LIN {X 0,Y 143.297,Z 453.566,A -85,B 0,C 180,E1 -24317.114,E2 -24317.114} C_VEL
LIN {X 0,Y 143.279,Z 453.631,A -85,B 0,C 180,E1 -24321.255,E2 -24321.255} C_VEL
LIN {X 0,Y 143.191,Z 453.587,A -85,B 0,C 180,E1 -24327.936,E2 -24327.936} C_VEL
LIN {X 0,Y 143.153,Z 453.64,A -85,B 0,C 180,E1 -24331.545,E2 -24331.545} C_VEL
LIN {X 0,Y 144.077,Z 456.331,A -85,B 0,C 180,E1 -24332.694,E2 -24332.694} C_VEL
LIN {X 0,Y 146.083,Z 458.522,A -85,B 0,C 180,E1 -24334.465,E2 -24334.465} C_VEL
LIN {X 0,Y 146.787,Z 459.324,A -85,B 0,C 180,E1 -24335.068,E2 -24335.068} C_VEL
LIN {X 0,Y 148.061,Z 461.946,A -85,B 0,C 180,E1 -24336.393,E2 -24336.393} C_VEL
LIN {X 0,Y 149.588,Z 463.631,A -85,B 0,C 180,E1 -24337.646,E2 -24337.646} C_VEL
LIN {X 0,Y 151.047,Z 466.609,A -85,B 0,C 180,E1 -24339.128,E2 -24339.128} C_VEL
LIN {X 0,Y 154.334,Z 472.293,A -85,B 0,C 180,E1 -24342.197,E2 -24342.197} C_VEL
LIN {X 0,Y 157.932,Z 480.262,A -85,B 0,C 180,E1 -24346.023,E2 -24346.023} C_VEL
LIN {X 0,Y 160.847,Z 488.732,A -85,B 0,C 180,E1 -24349.874,E2 -24349.874} C_VEL
LIN {X 0,Y 162.593,Z 495.92,A -85,B 0,C 180,E1 -24353.096,E2 -24353.096} C_VEL
LIN {X 0,Y 163.683,Z 502.348,A -85,B 0,C 180,E1 -24356.07,E2 -24356.07} C_VEL
LIN {X 0,Y 163.818,Z 503.973,A -85,B 0,C 180,E1 -24356.839,E2 -24356.839} C_VEL
LIN {X 0,Y 161.807,Z 508.944,A -85,B 0,C 180,E1 -24358.586,E2 -24358.586} C_VEL
LIN {X 0,Y 157.646,Z 517.43,A -85,B 0,C 180,E1 -24362.089,E2 -24362.089} C_VEL
LIN {X 0,Y 153.752,Z 524.699,A -85,B 0,C 180,E1 -24366.093,E2 -24366.093} C_VEL
LIN {X 0,Y 151.144,Z 529.533,A -85,B 0,C 180,E1 -24369.589,E2 -24369.589} C_VEL
LIN {X 0,Y 148.515,Z 533.769,A -85,B 0,C 180,E1 -24373.505,E2 -24373.505} C_VEL
LIN {X 0,Y 147.12,Z 536.002,A -85,B 0,C 180,E1 -24376.181,E2 -24376.181} C_VEL
LIN {X 0,Y 145.943,Z 537.821,A -85,B 0,C 180,E1 -24378.894,E2 -24378.894} C_VEL
LIN {X 0,Y 145.02,Z 539.188,A -85,B 0,C 180,E1 -24381.64,E2 -24381.64} C_VEL
LIN {X 0,Y 144.307,Z 540.706,A -85,B 0,C 180,E1 -24387.208,E2 -24387.208} C_VEL
LIN {X 0,Y 144.213,Z 540.925,A -85,B 0,C 180,E1 -24390,E2 -24390} C_VEL
LIN {X 0,Y 144.306,Z 540.736,A -85,B 0,C 180,E1 -24392.791,E2 -24392.791} C_VEL
LIN {X 0,Y 145.009,Z 539.256,A -85,B 0,C 180,E1 -24398.36,E2 -24398.36} C_VEL
LIN {X 0,Y 145.924,Z 537.921,A -85,B 0,C 180,E1 -24401.107,E2 -24401.107} C_VEL
LIN {X 0,Y 147.831,Z 535.093,A -85,B 0,C 180,E1 -24405.157,E2 -24405.157} C_VEL
LIN {X 0,Y 150.232,Z 531.269,A -85,B 0,C 180,E1 -24409.115,E2 -24409.115} C_VEL
LIN {X 0,Y 153.482,Z 525.332,A -85,B 0,C 180,E1 -24413.679,E2 -24413.679} C_VEL
LIN {X 0,Y 157.622,Z 517.742,A -85,B 0,C 180,E1 -24417.915,E2 -24417.915} C_VEL
LIN {X 0,Y 161.738,Z 509.36,A -85,B 0,C 180,E1 -24421.429,E2 -24421.429} C_VEL
LIN {X 0,Y 163.827,Z 504.413,A -85,B 0,C 180,E1 -24423.159,E2 -24423.159} C_VEL
LIN {X 0,Y 163.074,Z 497.829,A -85,B 0,C 180,E1 -24426.2,E2 -24426.2} C_VEL
LIN {X 0,Y 161.008,Z 488.99,A -85,B 0,C 180,E1 -24430.194,E2 -24430.194} C_VEL
LIN {X 0,Y 158.209,Z 480.766,A -85,B 0,C 180,E1 -24433.939,E2 -24433.939} C_VEL
LIN {X 0,Y 154.527,Z 472.644,A -85,B 0,C 180,E1 -24437.868,E2 -24437.868} C_VEL
LIN {X 0,Y 149.779,Z 464.121,A -85,B 0,C 180,E1 -24442.411,E2 -24442.411} C_VEL
LIN {X 0,Y 147.619,Z 461.218,A -85,B 0,C 180,E1 -24444.324,E2 -24444.324} C_VEL
LIN {X 0,Y 146.552,Z 458.872,A -85,B 0,C 180,E1 -24445.463,E2 -24445.463} C_VEL
LIN {X 0,Y 144.33,Z 456.714,A -85,B 0,C 180,E1 -24447.371,E2 -24447.371} C_VEL
LIN {X 0,Y 143.255,Z 454.252,A -85,B 0,C 180,E1 -24448.583,E2 -24448.583} C_VEL
LIN {X 0,Y 143.158,Z 453.648,A -85,B 0,C 180,E1 -24448.868,E2 -24448.868} C_VEL
LIN {X 0,Y 143.161,Z 453.647,A -85,B 0,C 180,E1 -24453.779,E2 -24453.779} C_VEL
LIN {X 0,Y 143.311,Z 453.634,A -85,B 0,C 180,E1 -24459.923,E2 -24459.923} C_VEL
LIN {X 0,Y 143.364,Z 453.627,A -85,B 0,C 180,E1 -24465.811,E2 -24465.811} C_VEL
LIN {X 0,Y 143.539,Z 453.594,A -85,B 0,C 180,E1 -24468.705,E2 -24468.705} C_VEL
LIN {X 0,Y 143.627,Z 453.594,A -85,B 0,C 180,E1 -24471.558,E2 -24471.558} C_VEL
LIN {X 0,Y 144.179,Z 453.515,A -85,B 0,C 180,E1 -24480,E2 -24480} C_VEL
LIN {X 0,Y 143.627,Z 453.581,A -85,B 0,C 180,E1 -24488.441,E2 -24488.441} C_VEL
LIN {X 0,Y 143.507,Z 453.601,A -85,B 0,C 180,E1 -24491.631,E2 -24491.631} C_VEL
LIN {X 0,Y 143.349,Z 453.727,A -85,B 0,C 180,E1 -24494.552,E2 -24494.552} C_VEL
LIN {X 0,Y 143.984,Z 456.816,A -85,B 0,C 180,E1 -24499.979,E2 -24499.979} C_VEL
LIN {X 0,Y 145.063,Z 461.745,A -85,B 0,C 180,E1 -24507.404,E2 -24507.404} C_VEL
LIN {X 0,Y 145.674,Z 465.026,A -85,B 0,C 180,E1 -24511.456,E2 -24511.456} C_VEL
LIN {X 0,Y 147.336,Z 468.84,A -85,B 0,C 180,E1 -24512.86,E2 -24512.86} C_VEL
LIN {X 0,Y 149.667,Z 472.325,A -85,B 0,C 180,E1 -24514.58,E2 -24514.58} C_VEL
LIN {X 0,Y 151.366,Z 476.461,A -85,B 0,C 180,E1 -24515.989,E2 -24515.989} C_VEL
LIN {X 0,Y 152.885,Z 479.225,A -85,B 0,C 180,E1 -24517.11,E2 -24517.11} C_VEL
LIN {X 0,Y 155.096,Z 484.217,A -85,B 0,C 180,E1 -24518.852,E2 -24518.852} C_VEL
LIN {X 0,Y 159.394,Z 496.028,A -85,B 0,C 180,E1 -24522.582,E2 -24522.582} C_VEL
LIN {X 0,Y 159.768,Z 503.297,A -85,B 0,C 180,E1 -24524.191,E2 -24524.191} C_VEL
LIN {X 0,Y 159.384,Z 515.58,A -85,B 0,C 180,E1 -24527.018,E2 -24527.018} C_VEL
LIN {X 0,Y 158.225,Z 526.386,A -85,B 0,C 180,E1 -24529.818,E2 -24529.818} C_VEL
LIN {X 0,Y 156.296,Z 537.075,A -85,B 0,C 180,E1 -24533.028,E2 -24533.028} C_VEL
LIN {X 0,Y 154.059,Z 545.932,A -85,B 0,C 180,E1 -24536.151,E2 -24536.151} C_VEL
LIN {X 0,Y 151.298,Z 555.019,A -85,B 0,C 180,E1 -24540.043,E2 -24540.043} C_VEL
LIN {X 0,Y 148.719,Z 561.324,A -85,B 0,C 180,E1 -24543.324,E2 -24543.324} C_VEL
LIN {X 0,Y 145.685,Z 567.48,A -85,B 0,C 180,E1 -24547.299,E2 -24547.299} C_VEL
LIN {X 0,Y 143.571,Z 572.416,A -85,B 0,C 180,E1 -24551.447,E2 -24551.447} C_VEL
LIN {X 0,Y 142.375,Z 576.263,A -85,B 0,C 180,E1 -24555.711,E2 -24555.711} C_VEL
LIN {X 0,Y 142.003,Z 578.283,A -85,B 0,C 180,E1 -24558.582,E2 -24558.582} C_VEL
LIN {X 0,Y 142.305,Z 580.995,A -85,B 0,C 180,E1 -24564.332,E2 -24564.332} C_VEL
LIN {X 0,Y 142.75,Z 581.734,A -85,B 0,C 180,E1 -24567.178,E2 -24567.178} C_VEL
LIN {X 0,Y 143.416,Z 582.062,A -85,B 0,C 180,E1 -24570,E2 -24570} C_VEL
LIN {X 0,Y 142.744,Z 581.719,A -85,B 0,C 180,E1 -24572.822,E2 -24572.822} C_VEL
LIN {X 0,Y 142.297,Z 580.972,A -85,B 0,C 180,E1 -24575.669,E2 -24575.669} C_VEL
LIN {X 0,Y 142.004,Z 579.81,A -85,B 0,C 180,E1 -24578.539,E2 -24578.539} C_VEL
LIN {X 0,Y 142.155,Z 577.262,A -85,B 0,C 180,E1 -24582.855,E2 -24582.855} C_VEL
LIN {X 0,Y 143.044,Z 573.723,A -85,B 0,C 180,E1 -24587.145,E2 -24587.145} C_VEL
LIN {X 0,Y 144.83,Z 569.135,A -85,B 0,C 180,E1 -24591.343,E2 -24591.343} C_VEL
LIN {X 0,Y 148.156,Z 562.333,A -85,B 0,C 180,E1 -24596.027,E2 -24596.027} C_VEL
LIN {X 0,Y 150.773,Z 556.234,A -85,B 0,C 180,E1 -24599.304,E2 -24599.304} C_VEL
LIN {X 0,Y 153.633,Z 547.156,A -85,B 0,C 180,E1 -24603.295,E2 -24603.295} C_VEL
LIN {X 0,Y 156,Z 537.835,A -85,B 0,C 180,E1 -24606.651,E2 -24606.651} C_VEL
LIN {X 0,Y 157.978,Z 527.397,A -85,B 0,C 180,E1 -24609.814,E2 -24609.814} C_VEL
LIN {X 0,Y 159.187,Z 516.722,A -85,B 0,C 180,E1 -24612.626,E2 -24612.626} C_VEL
LIN {X 0,Y 159.693,Z 504.397,A -85,B 0,C 180,E1 -24615.481,E2 -24615.481} C_VEL
LIN {X 0,Y 159.493,Z 497.348,A -85,B 0,C 180,E1 -24617.002,E2 -24617.002} C_VEL
LIN {X 0,Y 158.812,Z 494.119,A -85,B 0,C 180,E1 -24617.868,E2 -24617.868} C_VEL
LIN {X 0,Y 154.735,Z 483.639,A -85,B 0,C 180,E1 -24621.249,E2 -24621.249} C_VEL
LIN {X 0,Y 153.2,Z 480.223,A -85,B 0,C 180,E1 -24622.45,E2 -24622.45} C_VEL
LIN {X 0,Y 152.039,Z 477.482,A -85,B 0,C 180,E1 -24623.379,E2 -24623.379} C_VEL
LIN {X 0,Y 150.429,Z 475.392,A -85,B 0,C 180,E1 -24624.466,E2 -24624.466} C_VEL
LIN {X 0,Y 146.597,Z 472.525,A -85,B 0,C 180,E1 -24626.916,E2 -24626.916} C_VEL
LIN {X 0,Y 142.658,Z 470.103,A -85,B 0,C 180,E1 -24629.618,E2 -24629.618} C_VEL
LIN {X 0,Y 140.203,Z 467.568,A -85,B 0,C 180,E1 -24631.637,E2 -24631.637} C_VEL
LIN {X 0,Y 139.55,Z 466.445,A -85,B 0,C 180,E1 -24632.278,E2 -24632.278} C_VEL
LIN {X 0,Y 137.989,Z 462.532,A -85,B 0,C 180,E1 -24634.145,E2 -24634.145} C_VEL
LIN {X 0,Y 137.296,Z 459.461,A -85,B 0,C 180,E1 -24639.003,E2 -24639.003} C_VEL
LIN {X 0,Y 136.944,Z 457.668,A -85,B 0,C 180,E1 -24642.066,E2 -24642.066} C_VEL
LIN {X 0,Y 136.47,Z 454.488,A -85,B 0,C 180,E1 -24648.387,E2 -24648.387} C_VEL
LIN {X 0,Y 136.554,Z 454.477,A -85,B 0,C 180,E1 -24651.118,E2 -24651.118} C_VEL
LIN {X 0,Y 137.137,Z 454.4,A -85,B 0,C 180,E1 -24660,E2 -24660} C_VEL
LIN {X 0,Y 136.554,Z 454.476,A -85,B 0,C 180,E1 -24668.882,E2 -24668.882} C_VEL
LIN {X 0,Y 136.443,Z 454.448,A -85,B 0,C 180,E1 -24671.89,E2 -24671.89} C_VEL
LIN {X 0,Y 136.215,Z 454.454,A -85,B 0,C 180,E1 -24678.034,E2 -24678.034} C_VEL
LIN {X 0,Y 136.2,Z 454.515,A -85,B 0,C 180,E1 -24681.749,E2 -24681.749} C_VEL
LIN {X 0,Y 136.123,Z 454.518,A -85,B 0,C 180,E1 -24686.031,E2 -24686.031} C_VEL
LIN {X 0,Y 136.969,Z 457.004,A -85,B 0,C 180,E1 -24687.4,E2 -24687.4} C_VEL
LIN {X 0,Y 138.795,Z 459.225,A -85,B 0,C 180,E1 -24689.47,E2 -24689.47} C_VEL
LIN {X 0,Y 139.999,Z 460.171,A -85,B 0,C 180,E1 -24690.654,E2 -24690.654} C_VEL
LIN {X 0,Y 141.216,Z 462.885,A -85,B 0,C 180,E1 -24692.214,E2 -24692.214} C_VEL
LIN {X 0,Y 143.317,Z 465.418,A -85,B 0,C 180,E1 -24694.329,E2 -24694.329} C_VEL
LIN {X 0,Y 144.49,Z 467.805,A -85,B 0,C 180,E1 -24695.71,E2 -24695.71} C_VEL
LIN {X 0,Y 145.415,Z 468.906,A -85,B 0,C 180,E1 -24696.586,E2 -24696.586} C_VEL
LIN {X 0,Y 150.05,Z 477.982,A -85,B 0,C 180,E1 -24701.779,E2 -24701.779} C_VEL
LIN {X 0,Y 152.992,Z 485.164,A -85,B 0,C 180,E1 -24705.508,E2 -24705.508} C_VEL
LIN {X 0,Y 155.326,Z 492.952,A -85,B 0,C 180,E1 -24709.323,E2 -24709.323} C_VEL
LIN {X 0,Y 156.807,Z 500.167,A -85,B 0,C 180,E1 -24712.836,E2 -24712.836} C_VEL
LIN {X 0,Y 157.46,Z 505.072,A -85,B 0,C 180,E1 -24715.314,E2 -24715.314} C_VEL
LIN {X 0,Y 157.385,Z 506.694,A -85,B 0,C 180,E1 -24716.069,E2 -24716.069} C_VEL
LIN {X 0,Y 153.607,Z 514.435,A -85,B 0,C 180,E1 -24719.021,E2 -24719.021} C_VEL
LIN {X 0,Y 149.493,Z 521.994,A -85,B 0,C 180,E1 -24722.718,E2 -24722.718} C_VEL
LIN {X 0,Y 146.667,Z 527.077,A -85,B 0,C 180,E1 -24725.932,E2 -24725.932} C_VEL
LIN {X 0,Y 143.655,Z 532.088,A -85,B 0,C 180,E1 -24729.973,E2 -24729.973} C_VEL
LIN {X 0,Y 141.075,Z 535.962,A -85,B 0,C 180,E1 -24734.097,E2 -24734.097} C_VEL
LIN {X 0,Y 139.053,Z 538.827,A -85,B 0,C 180,E1 -24738.336,E2 -24738.336} C_VEL
LIN {X 0,Y 138.07,Z 540.193,A -85,B 0,C 180,E1 -24741.216,E2 -24741.216} C_VEL
LIN {X 0,Y 137.288,Z 541.712,A -85,B 0,C 180,E1 -24747.065,E2 -24747.065} C_VEL
LIN {X 0,Y 137.186,Z 541.93,A -85,B 0,C 180,E1 -24750,E2 -24750} C_VEL
LIN {X 0,Y 137.287,Z 541.741,A -85,B 0,C 180,E1 -24752.934,E2 -24752.934} C_VEL
LIN {X 0,Y 138.059,Z 540.261,A -85,B 0,C 180,E1 -24758.784,E2 -24758.784} C_VEL
LIN {X 0,Y 139.034,Z 538.925,A -85,B 0,C 180,E1 -24761.665,E2 -24761.665} C_VEL
LIN {X 0,Y 141.06,Z 536.097,A -85,B 0,C 180,E1 -24765.904,E2 -24765.904} C_VEL
LIN {X 0,Y 143.61,Z 532.273,A -85,B 0,C 180,E1 -24770.033,E2 -24770.033} C_VEL
LIN {X 0,Y 147.073,Z 526.335,A -85,B 0,C 180,E1 -24774.779,E2 -24774.779} C_VEL
LIN {X 0,Y 151.448,Z 518.745,A -85,B 0,C 180,E1 -24779.16,E2 -24779.16} C_VEL
LIN {X 0,Y 155.787,Z 510.362,A -85,B 0,C 180,E1 -24782.776,E2 -24782.776} C_VEL
LIN {X 0,Y 157.316,Z 507.142,A -85,B 0,C 180,E1 -24783.947,E2 -24783.947} C_VEL
LIN {X 0,Y 157.546,Z 505.493,A -85,B 0,C 180,E1 -24784.664,E2 -24784.664} C_VEL
LIN {X 0,Y 156.753,Z 499.46,A -85,B 0,C 180,E1 -24787.7,E2 -24787.7} C_VEL
LIN {X 0,Y 155.031,Z 491.486,A -85,B 0,C 180,E1 -24791.583,E2 -24791.583} C_VEL
LIN {X 0,Y 153.006,Z 485.082,A -85,B 0,C 180,E1 -24794.754,E2 -24794.754} C_VEL
LIN {X 0,Y 149.992,Z 477.795,A -85,B 0,C 180,E1 -24798.564,E2 -24798.564} C_VEL
LIN {X 0,Y 146.032,Z 470.057,A -85,B 0,C 180,E1 -24803.018,E2 -24803.018} C_VEL
LIN {X 0,Y 143.522,Z 465.868,A -85,B 0,C 180,E1 -24805.727,E2 -24805.727} C_VEL
LIN {X 0,Y 140.452,Z 461.398,A -85,B 0,C 180,E1 -24809.037,E2 -24809.037} C_VEL
LIN {X 0,Y 139.876,Z 459.943,A -85,B 0,C 180,E1 -24809.838,E2 -24809.838} C_VEL
LIN {X 0,Y 137.633,Z 458.023,A -85,B 0,C 180,E1 -24812.159,E2 -24812.159} C_VEL
LIN {X 0,Y 136.391,Z 455.702,A -85,B 0,C 180,E1 -24813.818,E2 -24813.818} C_VEL
LIN {X 0,Y 136.11,Z 454.53,A -85,B 0,C 180,E1 -24814.48,E2 -24814.48} C_VEL
LIN {X 0,Y 136.246,Z 454.506,A -85,B 0,C 180,E1 -24818.833,E2 -24818.833} C_VEL
LIN {X 0,Y 136.274,Z 454.509,A -85,B 0,C 180,E1 -24825.056,E2 -24825.056} C_VEL
LIN {X 0,Y 136.446,Z 454.477,A -85,B 0,C 180,E1 -24828.138,E2 -24828.138} C_VEL
LIN {X 0,Y 136.553,Z 454.476,A -85,B 0,C 180,E1 -24831.118,E2 -24831.118} C_VEL
LIN {X 0,Y 137.136,Z 454.392,A -85,B 0,C 180,E1 -24840,E2 -24840} C_VEL
LIN {X 0,Y 136.553,Z 454.463,A -85,B 0,C 180,E1 -24848.882,E2 -24848.882} C_VEL
LIN {X 0,Y 136.459,Z 454.644,A -85,B 0,C 180,E1 -24851.889,E2 -24851.889} C_VEL
LIN {X 0,Y 136.954,Z 457.794,A -85,B 0,C 180,E1 -24857.933,E2 -24857.933} C_VEL
LIN {X 0,Y 137.658,Z 461.515,A -85,B 0,C 180,E1 -24864.106,E2 -24864.106} C_VEL
LIN {X 0,Y 137.986,Z 462.686,A -85,B 0,C 180,E1 -24865.755,E2 -24865.755} C_VEL
LIN {X 0,Y 139.872,Z 466.922,A -85,B 0,C 180,E1 -24867.797,E2 -24867.797} C_VEL
LIN {X 0,Y 142.506,Z 470.812,A -85,B 0,C 180,E1 -24870.205,E2 -24870.205} C_VEL
LIN {X 0,Y 144.675,Z 475.595,A -85,B 0,C 180,E1 -24872.3,E2 -24872.3} C_VEL
LIN {X 0,Y 145.984,Z 477.81,A -85,B 0,C 180,E1 -24873.41,E2 -24873.41} C_VEL
LIN {X 0,Y 148.138,Z 482.859,A -85,B 0,C 180,E1 -24875.429,E2 -24875.429} C_VEL
LIN {X 0,Y 152.267,Z 493.635,A -85,B 0,C 180,E1 -24879.393,E2 -24879.393} C_VEL
LIN {X 0,Y 154.104,Z 499.441,A -85,B 0,C 180,E1 -24881.362,E2 -24881.362} C_VEL
LIN {X 0,Y 154.051,Z 508.443,A -85,B 0,C 180,E1 -24883.509,E2 -24883.509} C_VEL
LIN {X 0,Y 153.152,Z 520.101,A -85,B 0,C 180,E1 -24886.502,E2 -24886.502} C_VEL
LIN {X 0,Y 151.471,Z 530.47,A -85,B 0,C 180,E1 -24889.49,E2 -24889.49} C_VEL
LIN {X 0,Y 149.045,Z 540.984,A -85,B 0,C 180,E1 -24893.054,E2 -24893.054} C_VEL
LIN {X 0,Y 146.412,Z 549.526,A -85,B 0,C 180,E1 -24896.494,E2 -24896.494} C_VEL
LIN {X 0,Y 143.945,Z 556.643,A -85,B 0,C 180,E1 -24899.97,E2 -24899.97} C_VEL
LIN {X 0,Y 141.209,Z 562.506,A -85,B 0,C 180,E1 -24903.389,E2 -24903.389} C_VEL
LIN {X 0,Y 138.208,Z 568.218,A -85,B 0,C 180,E1 -24907.581,E2 -24907.581} C_VEL
LIN {X 0,Y 136.211,Z 572.776,A -85,B 0,C 180,E1 -24911.966,E2 -24911.966} C_VEL
LIN {X 0,Y 135.168,Z 576.288,A -85,B 0,C 180,E1 -24916.469,E2 -24916.469} C_VEL
LIN {X 0,Y 134.957,Z 579.099,A -85,B 0,C 180,E1 -24921.667,E2 -24921.667} C_VEL
LIN {X 0,Y 135.667,Z 580.72,A -85,B 0,C 180,E1 -24927.031,E2 -24927.031} C_VEL
LIN {X 0,Y 136.333,Z 581.049,A -85,B 0,C 180,E1 -24930,E2 -24930} C_VEL
LIN {X 0,Y 135.66,Z 580.704,A -85,B 0,C 180,E1 -24932.97,E2 -24932.97} C_VEL
LIN {X 0,Y 134.96,Z 579.063,A -85,B 0,C 180,E1 -24938.342,E2 -24938.342} C_VEL
LIN {X 0,Y 135.168,Z 576.235,A -85,B 0,C 180,E1 -24943.532,E2 -24943.532} C_VEL
LIN {X 0,Y 136.2,Z 572.695,A -85,B 0,C 180,E1 -24948.036,E2 -24948.036} C_VEL
LIN {X 0,Y 138.184,Z 568.109,A -85,B 0,C 180,E1 -24952.424,E2 -24952.424} C_VEL
LIN {X 0,Y 141.208,Z 562.376,A -85,B 0,C 180,E1 -24956.612,E2 -24956.612} C_VEL
LIN {X 0,Y 143.929,Z 556.48,A -85,B 0,C 180,E1 -24960.034,E2 -24960.034} C_VEL
LIN {X 0,Y 146.964,Z 547.771,A -85,B 0,C 180,E1 -24964.188,E2 -24964.188} C_VEL
LIN {X 0,Y 149.519,Z 538.809,A -85,B 0,C 180,E1 -24967.666,E2 -24967.666} C_VEL
LIN {X 0,Y 151.741,Z 528.639,A -85,B 0,C 180,E1 -24970.972,E2 -24970.972} C_VEL
LIN {X 0,Y 153.311,Z 517.349,A -85,B 0,C 180,E1 -24974.149,E2 -24974.149} C_VEL
LIN {X 0,Y 154.053,Z 506.389,A -85,B 0,C 180,E1 -24976.881,E2 -24976.881} C_VEL
LIN {X 0,Y 154.082,Z 499.92,A -85,B 0,C 180,E1 -24978.402,E2 -24978.402} C_VEL
LIN {X 0,Y 152.762,Z 495.326,A -85,B 0,C 180,E1 -24979.903,E2 -24979.903} C_VEL
LIN {X 0,Y 150.122,Z 487.982,A -85,B 0,C 180,E1 -24982.512,E2 -24982.512} C_VEL
LIN {X 0,Y 147.883,Z 482.444,A -85,B 0,C 180,E1 -24984.605,E2 -24984.605} C_VEL
LIN {X 0,Y 145.909,Z 477.69,A -85,B 0,C 180,E1 -24986.467,E2 -24986.467} C_VEL
LIN {X 0,Y 142.985,Z 472.291,A -85,B 0,C 180,E1 -24989.065,E2 -24989.065} C_VEL
LIN {X 0,Y 142.099,Z 470.177,A -85,B 0,C 180,E1 -24989.941,E2 -24989.941} C_VEL
LIN {X 0,Y 139.55,Z 466.445,A -85,B 0,C 180,E1 -24992.278,E2 -24992.278} C_VEL
LIN {X 0,Y 138.114,Z 464.818,A -85,B 0,C 180,E1 -24993.627,E2 -24993.627} C_VEL
LIN {X 0,Y 135.241,Z 464.181,A -85,B 0,C 180,E1 -24996.151,E2 -24996.151} C_VEL
LIN {X 0,Y 132.495,Z 463.872,A -85,B 0,C 180,E1 -24998.842,E2 -24998.842} C_VEL
LIN {X 0,Y 131.229,Z 462.693,A -85,B 0,C 180,E1 -25000.433,E2 -25000.433} C_VEL
LIN {X 0,Y 130.171,Z 459.727,A -85,B 0,C 180,E1 -25002.32,E2 -25002.32} C_VEL
LIN {X 0,Y 129.74,Z 457.139,A -85,B 0,C 180,E1 -25007.486,E2 -25007.486} C_VEL
LIN {X 0,Y 129.5,Z 455.358,A -85,B 0,C 180,E1 -25011.81,E2 -25011.81} C_VEL
LIN {X 0,Y 130.092,Z 455.277,A -85,B 0,C 180,E1 -25020,E2 -25020} C_VEL
LIN {X 0,Y 129.476,Z 455.356,A -85,B 0,C 180,E1 -25029.372,E2 -25029.372} C_VEL
LIN {X 0,Y 129.346,Z 455.317,A -85,B 0,C 180,E1 -25032.553,E2 -25032.553} C_VEL
LIN {X 0,Y 129.188,Z 455.458,A -85,B 0,C 180,E1 -25038.229,E2 -25038.229} C_VEL
LIN {X 0,Y 129.837,Z 457.662,A -85,B 0,C 180,E1 -25039.877,E2 -25039.877} C_VEL
LIN {X 0,Y 132.116,Z 460.379,A -85,B 0,C 180,E1 -25043.514,E2 -25043.514} C_VEL
LIN {X 0,Y 133.397,Z 461.221,A -85,B 0,C 180,E1 -25045.157,E2 -25045.157} C_VEL
LIN {X 0,Y 134.207,Z 463.303,A -85,B 0,C 180,E1 -25046.599,E2 -25046.599} C_VEL
LIN {X 0,Y 135.155,Z 464.733,A -85,B 0,C 180,E1 -25047.905,E2 -25047.905} C_VEL
LIN {X 0,Y 136.344,Z 465.895,A -85,B 0,C 180,E1 -25049.32,E2 -25049.32} C_VEL
LIN {X 0,Y 139.676,Z 471.37,A -85,B 0,C 180,E1 -25053.606,E2 -25053.606} C_VEL
LIN {X 0,Y 143.304,Z 478.471,A -85,B 0,C 180,E1 -25058.308,E2 -25058.308} C_VEL
LIN {X 0,Y 146.235,Z 485.115,A -85,B 0,C 180,E1 -25062.286,E2 -25062.286} C_VEL
LIN {X 0,Y 148.581,Z 492.38,A -85,B 0,C 180,E1 -25066.272,E2 -25066.272} C_VEL
LIN {X 0,Y 150.046,Z 498.569,A -85,B 0,C 180,E1 -25069.563,E2 -25069.563} C_VEL
LIN {X 0,Y 151.11,Z 505.971,A -85,B 0,C 180,E1 -25073.516,E2 -25073.516} C_VEL
LIN {X 0,Y 151.261,Z 508.023,A -85,B 0,C 180,E1 -25074.627,E2 -25074.627} C_VEL
LIN {X 0,Y 150.003,Z 510.957,A -85,B 0,C 180,E1 -25075.789,E2 -25075.789} C_VEL
LIN {X 0,Y 145.377,Z 519.444,A -85,B 0,C 180,E1 -25079.495,E2 -25079.495} C_VEL
LIN {X 0,Y 141.017,Z 526.712,A -85,B 0,C 180,E1 -25083.778,E2 -25083.778} C_VEL
LIN {X 0,Y 138.061,Z 531.545,A -85,B 0,C 180,E1 -25087.555,E2 -25087.555} C_VEL
LIN {X 0,Y 135.097,Z 535.781,A -85,B 0,C 180,E1 -25091.812,E2 -25091.812} C_VEL
LIN {X 0,Y 133.514,Z 538.014,A -85,B 0,C 180,E1 -25094.74,E2 -25094.74} C_VEL
LIN {X 0,Y 132.178,Z 539.833,A -85,B 0,C 180,E1 -25097.72,E2 -25097.72} C_VEL
LIN {X 0,Y 131.129,Z 541.199,A -85,B 0,C 180,E1 -25100.747,E2 -25100.747} C_VEL
LIN {X 0,Y 130.27,Z 542.717,A -85,B 0,C 180,E1 -25106.907,E2 -25106.907} C_VEL
LIN {X 0,Y 130.158,Z 542.935,A -85,B 0,C 180,E1 -25110,E2 -25110} C_VEL
LIN {X 0,Y 130.268,Z 542.746,A -85,B 0,C 180,E1 -25113.092,E2 -25113.092} C_VEL
LIN {X 0,Y 131.118,Z 541.266,A -85,B 0,C 180,E1 -25119.253,E2 -25119.253} C_VEL
LIN {X 0,Y 132.159,Z 539.93,A -85,B 0,C 180,E1 -25122.281,E2 -25122.281} C_VEL
LIN {X 0,Y 134.315,Z 537.101,A -85,B 0,C 180,E1 -25126.725,E2 -25126.725} C_VEL
LIN {X 0,Y 137.029,Z 533.277,A -85,B 0,C 180,E1 -25131.04,E2 -25131.04} C_VEL
LIN {X 0,Y 140.72,Z 527.342,A -85,B 0,C 180,E1 -25135.976,E2 -25135.976} C_VEL
LIN {X 0,Y 144.655,Z 520.948,A -85,B 0,C 180,E1 -25139.867,E2 -25139.867} C_VEL
LIN {X 0,Y 149.151,Z 512.898,A -85,B 0,C 180,E1 -25143.618,E2 -25143.618} C_VEL
LIN {X 0,Y 151.324,Z 508.33,A -85,B 0,C 180,E1 -25145.412,E2 -25145.412} C_VEL
LIN {X 0,Y 150.675,Z 502.12,A -85,B 0,C 180,E1 -25148.774,E2 -25148.774} C_VEL
LIN {X 0,Y 149.565,Z 495.877,A -85,B 0,C 180,E1 -25152.059,E2 -25152.059} C_VEL
LIN {X 0,Y 147.352,Z 488.147,A -85,B 0,C 180,E1 -25156.242,E2 -25156.242} C_VEL
LIN {X 0,Y 144.829,Z 481.668,A -85,B 0,C 180,E1 -25159.986,E2 -25159.986} C_VEL
LIN {X 0,Y 141.538,Z 474.841,A -85,B 0,C 180,E1 -25164.307,E2 -25164.307} C_VEL
LIN {X 0,Y 138.953,Z 470.352,A -85,B 0,C 180,E1 -25167.564,E2 -25167.564} C_VEL
LIN {X 0,Y 136.479,Z 466.051,A -85,B 0,C 180,E1 -25170.881,E2 -25170.881} C_VEL
LIN {X 0,Y 134.091,Z 463.143,A -85,B 0,C 180,E1 -25173.963,E2 -25173.963} C_VEL
LIN {X 0,Y 133.266,Z 461.046,A -85,B 0,C 180,E1 -25175.461,E2 -25175.461} C_VEL
LIN {X 0,Y 130.936,Z 459.235,A -85,B 0,C 180,E1 -25178.681,E2 -25178.681} C_VEL
LIN {X 0,Y 129.523,Z 456.831,A -85,B 0,C 180,E1 -25181.411,E2 -25181.411} C_VEL
LIN {X 0,Y 129.182,Z 455.382,A -85,B 0,C 180,E1 -25182.385,E2 -25182.385} C_VEL
LIN {X 0,Y 129.368,Z 455.358,A -85,B 0,C 180,E1 -25187.922,E2 -25187.922} C_VEL
LIN {X 0,Y 129.478,Z 455.356,A -85,B 0,C 180,E1 -25190.628,E2 -25190.628} C_VEL
LIN {X 0,Y 130.091,Z 455.268,A -85,B 0,C 180,E1 -25200,E2 -25200} C_VEL
LIN {X 0,Y 129.53,Z 455.5,A -85,B 0,C 180,E1 -25208.581,E2 -25208.581} C_VEL
LIN {X 0,Y 129.75,Z 457.404,A -85,B 0,C 180,E1 -25212.844,E2 -25212.844} C_VEL
LIN {X 0,Y 130.149,Z 459.713,A -85,B 0,C 180,E1 -25217.277,E2 -25217.277} C_VEL
LIN {X 0,Y 131.805,Z 463.766,A -85,B 0,C 180,E1 -25220.075,E2 -25220.075} C_VEL
LIN {X 0,Y 135.35,Z 468.83,A -85,B 0,C 180,E1 -25224.544,E2 -25224.544} C_VEL
LIN {X 0,Y 137.298,Z 473.378,A -85,B 0,C 180,E1 -25227.019,E2 -25227.019} C_VEL
LIN {X 0,Y 139.247,Z 476.624,A -85,B 0,C 180,E1 -25229.064,E2 -25229.064} C_VEL
LIN {X 0,Y 141.464,Z 481.703,A -85,B 0,C 180,E1 -25231.547,E2 -25231.547} C_VEL
LIN {X 0,Y 142.062,Z 482.788,A -85,B 0,C 180,E1 -25232.128,E2 -25232.128} C_VEL
LIN {X 0,Y 146.152,Z 494.017,A -85,B 0,C 180,E1 -25236.803,E2 -25236.803} C_VEL
LIN {X 0,Y 148.754,Z 502.712,A -85,B 0,C 180,E1 -25240.072,E2 -25240.072} C_VEL
LIN {X 0,Y 148.232,Z 512.521,A -85,B 0,C 180,E1 -25242.619,E2 -25242.619} C_VEL
LIN {X 0,Y 146.919,Z 523.083,A -85,B 0,C 180,E1 -25245.593,E2 -25245.593} C_VEL
LIN {X 0,Y 144.737,Z 533.88,A -85,B 0,C 180,E1 -25249.041,E2 -25249.041} C_VEL
LIN {X 0,Y 141.833,Z 544.178,A -85,B 0,C 180,E1 -25252.96,E2 -25252.96} C_VEL
LIN {X 0,Y 138.701,Z 552.912,A -85,B 0,C 180,E1 -25256.996,E2 -25256.996} C_VEL
LIN {X 0,Y 136.055,Z 559.276,A -85,B 0,C 180,E1 -25260.612,E2 -25260.612} C_VEL
LIN {X 0,Y 132.608,Z 565.438,A -85,B 0,C 180,E1 -25264.914,E2 -25264.914} C_VEL
LIN {X 0,Y 130.075,Z 570.37,A -85,B 0,C 180,E1 -25269.44,E2 -25269.44} C_VEL
LIN {X 0,Y 128.498,Z 574.209,A -85,B 0,C 180,E1 -25274.13,E2 -25274.13} C_VEL
LIN {X 0,Y 127.983,Z 576.234,A -85,B 0,C 180,E1 -25277.312,E2 -25277.312} C_VEL
LIN {X 0,Y 127.914,Z 578.194,A -85,B 0,C 180,E1 -25281.486,E2 -25281.486} C_VEL
LIN {X 0,Y 128.58,Z 579.705,A -85,B 0,C 180,E1 -25286.867,E2 -25286.867} C_VEL
LIN {X 0,Y 129.248,Z 580.036,A -85,B 0,C 180,E1 -25290,E2 -25290} C_VEL
LIN {X 0,Y 128.574,Z 579.689,A -85,B 0,C 180,E1 -25293.134,E2 -25293.134} C_VEL
LIN {X 0,Y 127.915,Z 578.159,A -85,B 0,C 180,E1 -25298.518,E2 -25298.518} C_VEL
LIN {X 0,Y 128.218,Z 575.21,A -85,B 0,C 180,E1 -25304.28,E2 -25304.28} C_VEL
LIN {X 0,Y 129.399,Z 571.669,A -85,B 0,C 180,E1 -25309.019,E2 -25309.019} C_VEL
LIN {X 0,Y 131.602,Z 567.085,A -85,B 0,C 180,E1 -25313.612,E2 -25313.612} C_VEL
LIN {X 0,Y 135.449,Z 560.284,A -85,B 0,C 180,E1 -25318.683,E2 -25318.683} C_VEL
LIN {X 0,Y 138.176,Z 554.133,A -85,B 0,C 180,E1 -25322.281,E2 -25322.281} C_VEL
LIN {X 0,Y 140.902,Z 546.71,A -85,B 0,C 180,E1 -25325.879,E2 -25325.879} C_VEL
LIN {X 0,Y 143.607,Z 537.725,A -85,B 0,C 180,E1 -25329.51,E2 -25329.51} C_VEL
LIN {X 0,Y 145.958,Z 527.934,A -85,B 0,C 180,E1 -25332.824,E2 -25332.824} C_VEL
LIN {X 0,Y 147.707,Z 516.617,A -85,B 0,C 180,E1 -25336.169,E2 -25336.169} C_VEL
LIN {X 0,Y 148.653,Z 505.228,A -85,B 0,C 180,E1 -25339.153,E2 -25339.153} C_VEL
LIN {X 0,Y 148.644,Z 502.462,A -85,B 0,C 180,E1 -25339.892,E2 -25339.892} C_VEL
LIN {X 0,Y 146.131,Z 494.096,A -85,B 0,C 180,E1 -25343.026,E2 -25343.026} C_VEL
LIN {X 0,Y 142.737,Z 485.007,A -85,B 0,C 180,E1 -25346.829,E2 -25346.829} C_VEL
LIN {X 0,Y 141.534,Z 481.965,A -85,B 0,C 180,E1 -25348.157,E2 -25348.157} C_VEL
LIN {X 0,Y 139.278,Z 476.936,A -85,B 0,C 180,E1 -25350.632,E2 -25350.632} C_VEL
LIN {X 0,Y 138.479,Z 475.365,A -85,B 0,C 180,E1 -25351.486,E2 -25351.486} C_VEL
LIN {X 0,Y 136.03,Z 470.772,A -85,B 0,C 180,E1 -25354.259,E2 -25354.259} C_VEL
LIN {X 0,Y 135.148,Z 468.477,A -85,B 0,C 180,E1 -25355.417,E2 -25355.417} C_VEL
LIN {X 0,Y 132.023,Z 464.207,A -85,B 0,C 180,E1 -25359.247,E2 -25359.247} C_VEL
LIN {X 0,Y 131.229,Z 462.693,A -85,B 0,C 180,E1 -25360.433,E2 -25360.433} C_VEL
LIN {X 0,Y 129.628,Z 460.811,A -85,B 0,C 180,E1 -25362.78,E2 -25362.78} C_VEL
LIN {X 0,Y 127.982,Z 460.108,A -85,B 0,C 180,E1 -25365.3,E2 -25365.3} C_VEL
LIN {X 0,Y 124.458,Z 460.178,A -85,B 0,C 180,E1 -25372.467,E2 -25372.467} C_VEL
LIN {X 0,Y 123.954,Z 459.792,A -85,B 0,C 180,E1 -25374.312,E2 -25374.312} C_VEL
LIN {X 0,Y 123.409,Z 457.667,A -85,B 0,C 180,E1 -25380,E2 -25380} C_VEL
LIN {X 0,Y 125.062,Z 460.981,A -85,B 0,C 180,E1 -25392.99,E2 -25392.99} C_VEL
LIN {X 0,Y 127.004,Z 462.344,A -85,B 0,C 180,E1 -25397.408,E2 -25397.408} C_VEL
LIN {X 0,Y 127.975,Z 464.951,A -85,B 0,C 180,E1 -25400.074,E2 -25400.074} C_VEL
LIN {X 0,Y 129.277,Z 466.622,A -85,B 0,C 180,E1 -25402.453,E2 -25402.453} C_VEL
LIN {X 0,Y 130.223,Z 467.325,A -85,B 0,C 180,E1 -25403.875,E2 -25403.875} C_VEL
LIN {X 0,Y 132.159,Z 471.036,A -85,B 0,C 180,E1 -25407.345,E2 -25407.345} C_VEL
LIN {X 0,Y 132.944,Z 471.847,A -85,B 0,C 180,E1 -25408.41,E2 -25408.41} C_VEL
LIN {X 0,Y 135.859,Z 477.197,A -85,B 0,C 180,E1 -25412.9,E2 -25412.9} C_VEL
LIN {X 0,Y 138.776,Z 483.492,A -85,B 0,C 180,E1 -25417.425,E2 -25417.425} C_VEL
LIN {X 0,Y 141.111,Z 489.407,A -85,B 0,C 180,E1 -25421.294,E2 -25421.294} C_VEL
LIN {X 0,Y 143.073,Z 496.247,A -85,B 0,C 180,E1 -25425.383,E2 -25425.383} C_VEL
LIN {X 0,Y 144.427,Z 503.416,A -85,B 0,C 180,E1 -25429.521,E2 -25429.521} C_VEL
LIN {X 0,Y 145.018,Z 509.554,A -85,B 0,C 180,E1 -25433.089,E2 -25433.089} C_VEL
LIN {X 0,Y 144.925,Z 510.712,A -85,B 0,C 180,E1 -25433.74,E2 -25433.74} C_VEL
LIN {X 0,Y 140.143,Z 519.142,A -85,B 0,C 180,E1 -25437.377,E2 -25437.377} C_VEL
LIN {X 0,Y 135.787,Z 526.181,A -85,B 0,C 180,E1 -25441.395,E2 -25441.395} C_VEL
LIN {X 0,Y 132.696,Z 530.903,A -85,B 0,C 180,E1 -25444.931,E2 -25444.931} C_VEL
LIN {X 0,Y 129.455,Z 535.495,A -85,B 0,C 180,E1 -25449.336,E2 -25449.336} C_VEL
LIN {X 0,Y 126.747,Z 539.02,A -85,B 0,C 180,E1 -25453.904,E2 -25453.904} C_VEL
LIN {X 0,Y 125.32,Z 540.839,A -85,B 0,C 180,E1 -25457.037,E2 -25457.037} C_VEL
LIN {X 0,Y 124.198,Z 542.205,A -85,B 0,C 180,E1 -25460.226,E2 -25460.226} C_VEL
LIN {X 0,Y 123.253,Z 543.722,A -85,B 0,C 180,E1 -25466.731,E2 -25466.731} C_VEL
LIN {X 0,Y 123.131,Z 543.94,A -85,B 0,C 180,E1 -25470,E2 -25470} C_VEL
LIN {X 0,Y 123.251,Z 543.751,A -85,B 0,C 180,E1 -25473.269,E2 -25473.269} C_VEL
LIN {X 0,Y 124.186,Z 542.27,A -85,B 0,C 180,E1 -25479.775,E2 -25479.775} C_VEL
LIN {X 0,Y 125.3,Z 540.935,A -85,B 0,C 180,E1 -25482.965,E2 -25482.965} C_VEL
LIN {X 0,Y 127.6,Z 538.106,A -85,B 0,C 180,E1 -25487.634,E2 -25487.634} C_VEL
LIN {X 0,Y 130.493,Z 534.281,A -85,B 0,C 180,E1 -25492.148,E2 -25492.148} C_VEL
LIN {X 0,Y 134.435,Z 528.349,A -85,B 0,C 180,E1 -25497.285,E2 -25497.285} C_VEL
LIN {X 0,Y 138.605,Z 521.951,A -85,B 0,C 180,E1 -25501.314,E2 -25501.314} C_VEL
LIN {X 0,Y 143.356,Z 513.901,A -85,B 0,C 180,E1 -25505.173,E2 -25505.173} C_VEL
LIN {X 0,Y 144.879,Z 511.067,A -85,B 0,C 180,E1 -25506.297,E2 -25506.297} C_VEL
LIN {X 0,Y 145.129,Z 509.85,A -85,B 0,C 180,E1 -25506.927,E2 -25506.927} C_VEL
LIN {X 0,Y 144.404,Z 502.8,A -85,B 0,C 180,E1 -25511.06,E2 -25511.06} C_VEL
LIN {X 0,Y 143.064,Z 495.812,A -85,B 0,C 180,E1 -25515.086,E2 -25515.086} C_VEL
LIN {X 0,Y 141.265,Z 489.725,A -85,B 0,C 180,E1 -25518.761,E2 -25518.761} C_VEL
LIN {X 0,Y 138.956,Z 483.796,A -85,B 0,C 180,E1 -25522.632,E2 -25522.632} C_VEL
LIN {X 0,Y 136.052,Z 477.558,A -85,B 0,C 180,E1 -25527.153,E2 -25527.153} C_VEL
LIN {X 0,Y 133.181,Z 472.142,A -85,B 0,C 180,E1 -25531.645,E2 -25531.645} C_VEL
LIN {X 0,Y 131.214,Z 469.486,A -85,B 0,C 180,E1 -25534.628,E2 -25534.628} C_VEL
LIN {X 0,Y 130.271,Z 467.376,A -85,B 0,C 180,E1 -25536.511,E2 -25536.511} C_VEL
LIN {X 0,Y 127.694,Z 464.407,A -85,B 0,C 180,E1 -25541.134,E2 -25541.134} C_VEL
LIN {X 0,Y 126.9,Z 462.102,A -85,B 0,C 180,E1 -25543.511,E2 -25543.511} C_VEL
LIN {X 0,Y 123.524,Z 458.568,A -85,B 0,C 180,E1 -25558.37,E2 -25558.37} C_VEL
LIN {X 0,Y 123.626,Z 458.412,A -85,B 0,C 180,E1 -25560.407,E2 -25560.407} C_VEL
LIN {X 0,Y 125.027,Z 461.114,A -85,B 0,C 180,E1 -25568.689,E2 -25568.689} C_VEL
LIN {X 0,Y 128.158,Z 466.275,A -85,B 0,C 180,E1 -25576.22,E2 -25576.22} C_VEL
LIN {X 0,Y 129.6,Z 470.236,A -85,B 0,C 180,E1 -25579.193,E2 -25579.193} C_VEL
LIN {X 0,Y 132.526,Z 475.011,A -85,B 0,C 180,E1 -25583.436,E2 -25583.436} C_VEL
LIN {X 0,Y 134.719,Z 480.244,A -85,B 0,C 180,E1 -25586.636,E2 -25586.636} C_VEL
LIN {X 0,Y 135.673,Z 482.018,A -85,B 0,C 180,E1 -25587.788,E2 -25587.788} C_VEL
LIN {X 0,Y 138.332,Z 489.035,A -85,B 0,C 180,E1 -25591.383,E2 -25591.383} C_VEL
LIN {X 0,Y 140.939,Z 496.905,A -85,B 0,C 180,E1 -25594.991,E2 -25594.991} C_VEL
LIN {X 0,Y 143.285,Z 505.636,A -85,B 0,C 180,E1 -25598.621,E2 -25598.621} C_VEL
LIN {X 0,Y 143.123,Z 509.801,A -85,B 0,C 180,E1 -25599.835,E2 -25599.835} C_VEL
LIN {X 0,Y 141.551,Z 521.369,A -85,B 0,C 180,E1 -25603.197,E2 -25603.197} C_VEL
LIN {X 0,Y 139.32,Z 531.687,A -85,B 0,C 180,E1 -25606.582,E2 -25606.582} C_VEL
LIN {X 0,Y 136.785,Z 540.51,A -85,B 0,C 180,E1 -25609.945,E2 -25609.945} C_VEL
LIN {X 0,Y 133.742,Z 548.981,A -85,B 0,C 180,E1 -25613.76,E2 -25613.76} C_VEL
LIN {X 0,Y 130.356,Z 557.068,A -85,B 0,C 180,E1 -25618.288,E2 -25618.288} C_VEL
LIN {X 0,Y 127.371,Z 562.489,A -85,B 0,C 180,E1 -25621.987,E2 -25621.987} C_VEL
LIN {X 0,Y 124.154,Z 567.832,A -85,B 0,C 180,E1 -25626.656,E2 -25626.656} C_VEL
LIN {X 0,Y 122.078,Z 572.031,A -85,B 0,C 180,E1 -25631.541,E2 -25631.541} C_VEL
LIN {X 0,Y 121.019,Z 575.212,A -85,B 0,C 180,E1 -25636.568,E2 -25636.568} C_VEL
LIN {X 0,Y 120.983,Z 577.929,A -85,B 0,C 180,E1 -25643.328,E2 -25643.328} C_VEL
LIN {X 0,Y 121.49,Z 578.689,A -85,B 0,C 180,E1 -25646.684,E2 -25646.684} C_VEL
LIN {X 0,Y 122.163,Z 579.022,A -85,B 0,C 180,E1 -25650,E2 -25650} C_VEL
LIN {X 0,Y 121.485,Z 578.673,A -85,B 0,C 180,E1 -25653.317,E2 -25653.317} C_VEL
LIN {X 0,Y 120.859,Z 577.268,A -85,B 0,C 180,E1 -25658.675,E2 -25658.675} C_VEL
LIN {X 0,Y 121.257,Z 574.18,A -85,B 0,C 180,E1 -25665.119,E2 -25665.119} C_VEL
LIN {X 0,Y 122.65,Z 570.643,A -85,B 0,C 180,E1 -25670.109,E2 -25670.109} C_VEL
LIN {X 0,Y 125.088,Z 566.062,A -85,B 0,C 180,E1 -25674.922,E2 -25674.922} C_VEL
LIN {X 0,Y 128.554,Z 560.323,A -85,B 0,C 180,E1 -25679.474,E2 -25679.474} C_VEL
LIN {X 0,Y 131.45,Z 554.381,A -85,B 0,C 180,E1 -25683.232,E2 -25683.232} C_VEL
LIN {X 0,Y 134.933,Z 545.642,A -85,B 0,C 180,E1 -25687.735,E2 -25687.735} C_VEL
LIN {X 0,Y 137.828,Z 536.634,A -85,B 0,C 180,E1 -25691.521,E2 -25691.521} C_VEL
LIN {X 0,Y 140.125,Z 527.967,A -85,B 0,C 180,E1 -25694.602,E2 -25694.602} C_VEL
LIN {X 0,Y 142.046,Z 517.436,A -85,B 0,C 180,E1 -25697.916,E2 -25697.916} C_VEL
LIN {X 0,Y 143.267,Z 506.866,A -85,B 0,C 180,E1 -25700.878,E2 -25700.878} C_VEL
LIN {X 0,Y 142.784,Z 503.9,A -85,B 0,C 180,E1 -25701.957,E2 -25701.957} C_VEL
LIN {X 0,Y 140.268,Z 495.098,A -85,B 0,C 180,E1 -25705.69,E2 -25705.69} C_VEL
LIN {X 0,Y 137.642,Z 487.226,A -85,B 0,C 180,E1 -25709.296,E2 -25709.296} C_VEL
LIN {X 0,Y 135.913,Z 483.087,A -85,B 0,C 180,E1 -25711.531,E2 -25711.531} C_VEL
LIN {X 0,Y 135.122,Z 481.039,A -85,B 0,C 180,E1 -25712.614,E2 -25712.614} C_VEL
LIN {X 0,Y 132.851,Z 476.161,A -85,B 0,C 180,E1 -25715.692,E2 -25715.692} C_VEL
LIN {X 0,Y 132.062,Z 474.195,A -85,B 0,C 180,E1 -25716.891,E2 -25716.891} C_VEL
LIN {X 0,Y 129.137,Z 469.294,A -85,B 0,C 180,E1 -25721.25,E2 -25721.25} C_VEL
LIN {X 0,Y 127.872,Z 465.874,A -85,B 0,C 180,E1 -25723.845,E2 -25723.845} C_VEL
LIN {X 0,Y 124.602,Z 460.487,A -85,B 0,C 180,E1 -25731.894,E2 -25731.894} C_VEL
LIN {X 0,Y 123.954,Z 459.792,A -85,B 0,C 180,E1 -25734.312,E2 -25734.312} C_VEL
LIN {X 0,Y 123.557,Z 459.616,A -85,B 0,C 180,E1 -25736.123,E2 -25736.123} C_VEL
LIN {X 0,Y 123.161,Z 460.104,A -85,B 0,C 180,E1 -25737.932,E2 -25737.932} C_VEL
LIN {X 0,Y 122.452,Z 462.297,A -85,B 0,C 180,E1 -25741.496,E2 -25741.496} C_VEL
LIN {X 0,Y 121.988,Z 466.051,A -85,B 0,C 180,E1 -25746.932,E2 -25746.932} C_VEL
LIN {X 0,Y 122.188,Z 466.692,A -85,B 0,C 180,E1 -25748.804,E2 -25748.804} C_VEL
LIN {X 0,Y 124.529,Z 468.702,A -85,B 0,C 180,E1 -25756.391,E2 -25756.391} C_VEL
LIN {X 0,Y 125.471,Z 471.529,A -85,B 0,C 180,E1 -25759.638,E2 -25759.638} C_VEL
LIN {X 0,Y 127.01,Z 473.452,A -85,B 0,C 180,E1 -25762.789,E2 -25762.789} C_VEL
LIN {X 0,Y 129.352,Z 477.724,A -85,B 0,C 180,E1 -25767.505,E2 -25767.505} C_VEL
LIN {X 0,Y 132.267,Z 483.938,A -85,B 0,C 180,E1 -25773,E2 -25773} C_VEL
LIN {X 0,Y 134.376,Z 489.015,A -85,B 0,C 180,E1 -25776.975,E2 -25776.975} C_VEL
LIN {X 0,Y 136.317,Z 494.897,A -85,B 0,C 180,E1 -25781.097,E2 -25781.097} C_VEL
LIN {X 0,Y 137.844,Z 501.791,A -85,B 0,C 180,E1 -25785.545,E2 -25785.545} C_VEL
LIN {X 0,Y 138.641,Z 508.081,A -85,B 0,C 180,E1 -25789.498,E2 -25789.498} C_VEL
LIN {X 0,Y 138.835,Z 511.096,A -85,B 0,C 180,E1 -25791.413,E2 -25791.413} C_VEL
LIN {X 0,Y 138.62,Z 512.97,A -85,B 0,C 180,E1 -25792.526,E2 -25792.526} C_VEL
LIN {X 0,Y 133.459,Z 521.458,A -85,B 0,C 180,E1 -25796.431,E2 -25796.431} C_VEL
LIN {X 0,Y 128.641,Z 528.628,A -85,B 0,C 180,E1 -25800.942,E2 -25800.942} C_VEL
LIN {X 0,Y 125.189,Z 533.557,A -85,B 0,C 180,E1 -25805.099,E2 -25805.099} C_VEL
LIN {X 0,Y 121.823,Z 537.794,A -85,B 0,C 180,E1 -25809.748,E2 -25809.748} C_VEL
LIN {X 0,Y 120.011,Z 540.026,A -85,B 0,C 180,E1 -25812.974,E2 -25812.974} C_VEL
LIN {X 0,Y 118.481,Z 541.844,A -85,B 0,C 180,E1 -25816.274,E2 -25816.274} C_VEL
LIN {X 0,Y 117.278,Z 543.21,A -85,B 0,C 180,E1 -25819.643,E2 -25819.643} C_VEL
LIN {X 0,Y 116.237,Z 544.728,A -85,B 0,C 180,E1 -25826.533,E2 -25826.533} C_VEL
LIN {X 0,Y 116.103,Z 544.945,A -85,B 0,C 180,E1 -25830,E2 -25830} C_VEL
LIN {X 0,Y 116.236,Z 544.756,A -85,B 0,C 180,E1 -25833.466,E2 -25833.466} C_VEL
LIN {X 0,Y 117.266,Z 543.275,A -85,B 0,C 180,E1 -25840.358,E2 -25840.358} C_VEL
LIN {X 0,Y 118.462,Z 541.939,A -85,B 0,C 180,E1 -25843.728,E2 -25843.728} C_VEL
LIN {X 0,Y 120.921,Z 539.11,A -85,B 0,C 180,E1 -25848.642,E2 -25848.642} C_VEL
LIN {X 0,Y 124.012,Z 535.285,A -85,B 0,C 180,E1 -25853.372,E2 -25853.372} C_VEL
LIN {X 0,Y 128.236,Z 529.345,A -85,B 0,C 180,E1 -25858.73,E2 -25858.73} C_VEL
LIN {X 0,Y 133.432,Z 521.754,A -85,B 0,C 180,E1 -25863.576,E2 -25863.576} C_VEL
LIN {X 0,Y 138.552,Z 513.365,A -85,B 0,C 180,E1 -25867.495,E2 -25867.495} C_VEL
LIN {X 0,Y 138.951,Z 511.386,A -85,B 0,C 180,E1 -25868.594,E2 -25868.594} C_VEL
LIN {X 0,Y 138.441,Z 505.017,A -85,B 0,C 180,E1 -25872.627,E2 -25872.627} C_VEL
LIN {X 0,Y 137.109,Z 497.694,A -85,B 0,C 180,E1 -25877.297,E2 -25877.297} C_VEL
LIN {X 0,Y 135.333,Z 491.602,A -85,B 0,C 180,E1 -25881.451,E2 -25881.451} C_VEL
LIN {X 0,Y 132.865,Z 485.202,A -85,B 0,C 180,E1 -25886.261,E2 -25886.261} C_VEL
LIN {X 0,Y 130.359,Z 479.769,A -85,B 0,C 180,E1 -25890.973,E2 -25890.973} C_VEL
LIN {X 0,Y 129.59,Z 477.975,A -85,B 0,C 180,E1 -25892.55,E2 -25892.55} C_VEL
LIN {X 0,Y 127.774,Z 474.915,A -85,B 0,C 180,E1 -25896.023,E2 -25896.023} C_VEL
LIN {X 0,Y 127.273,Z 473.68,A -85,B 0,C 180,E1 -25897.26,E2 -25897.26} C_VEL
LIN {X 0,Y 125.104,Z 470.717,A -85,B 0,C 180,E1 -25902.004,E2 -25902.004} C_VEL
LIN {X 0,Y 124.7,Z 469.252,A -85,B 0,C 180,E1 -25903.632,E2 -25903.632} C_VEL
LIN {X 0,Y 122.24,Z 466.703,A -85,B 0,C 180,E1 -25912.567,E2 -25912.567} C_VEL
LIN {X 0,Y 122.141,Z 465.275,A -85,B 0,C 180,E1 -25920,E2 -25920} C_VEL
LIN {X 0,Y 123.311,Z 467.803,A -85,B 0,C 180,E1 -25927.985,E2 -25927.985} C_VEL
LIN {X 0,Y 125.828,Z 472.557,A -85,B 0,C 180,E1 -25935.074,E2 -25935.074} C_VEL
LIN {X 0,Y 127.232,Z 476.93,A -85,B 0,C 180,E1 -25938.623,E2 -25938.623} C_VEL
LIN {X 0,Y 129.436,Z 480.989,A -85,B 0,C 180,E1 -25942.339,E2 -25942.339} C_VEL
LIN {X 0,Y 132.116,Z 487.968,A -85,B 0,C 180,E1 -25946.882,E2 -25946.882} C_VEL
LIN {X 0,Y 133.957,Z 493.382,A -85,B 0,C 180,E1 -25949.905,E2 -25949.905} C_VEL
LIN {X 0,Y 136.112,Z 501.109,A -85,B 0,C 180,E1 -25953.715,E2 -25953.715} C_VEL
LIN {X 0,Y 137.878,Z 508.906,A -85,B 0,C 180,E1 -25957.25,E2 -25957.25} C_VEL
LIN {X 0,Y 137.323,Z 514.008,A -85,B 0,C 180,E1 -25958.823,E2 -25958.823} C_VEL
LIN {X 0,Y 135.133,Z 525.555,A -85,B 0,C 180,E1 -25962.54,E2 -25962.54} C_VEL
LIN {X 0,Y 132.305,Z 535.831,A -85,B 0,C 180,E1 -25966.326,E2 -25966.326} C_VEL
LIN {X 0,Y 129.142,Z 544.788,A -85,B 0,C 180,E1 -25970.25,E2 -25970.25} C_VEL
LIN {X 0,Y 125.378,Z 553.502,A -85,B 0,C 180,E1 -25974.931,E2 -25974.931} C_VEL
LIN {X 0,Y 122.382,Z 559.439,A -85,B 0,C 180,E1 -25978.88,E2 -25978.88} C_VEL
LIN {X 0,Y 118.669,Z 565.155,A -85,B 0,C 180,E1 -25983.63,E2 -25983.63} C_VEL
LIN {X 0,Y 115.96,Z 569.704,A -85,B 0,C 180,E1 -25988.676,E2 -25988.676} C_VEL
LIN {X 0,Y 114.336,Z 573.209,A -85,B 0,C 180,E1 -25993.942,E2 -25993.942} C_VEL
LIN {X 0,Y 113.808,Z 576.407,A -85,B 0,C 180,E1 -26001.134,E2 -26001.134} C_VEL
LIN {X 0,Y 114.399,Z 577.674,A -85,B 0,C 180,E1 -26006.478,E2 -26006.478} C_VEL
LIN {X 0,Y 115.075,Z 578.008,A -85,B 0,C 180,E1 -26010,E2 -26010} C_VEL
LIN {X 0,Y 114.376,Z 577.655,A -85,B 0,C 180,E1 -26013.523,E2 -26013.523} C_VEL
LIN {X 0,Y 113.771,Z 575.714,A -85,B 0,C 180,E1 -26020.68,E2 -26020.68} C_VEL
LIN {X 0,Y 114.333,Z 573.151,A -85,B 0,C 180,E1 -26026.059,E2 -26026.059} C_VEL
LIN {X 0,Y 115.948,Z 569.617,A -85,B 0,C 180,E1 -26031.327,E2 -26031.327} C_VEL
LIN {X 0,Y 118.652,Z 565.04,A -85,B 0,C 180,E1 -26036.375,E2 -26036.375} C_VEL
LIN {X 0,Y 122.382,Z 559.3,A -85,B 0,C 180,E1 -26041.121,E2 -26041.121} C_VEL
LIN {X 0,Y 125.361,Z 553.327,A -85,B 0,C 180,E1 -26045.075,E2 -26045.075} C_VEL
LIN {X 0,Y 129.095,Z 544.569,A -85,B 0,C 180,E1 -26049.768,E2 -26049.768} C_VEL
LIN {X 0,Y 132.586,Z 534.519,A -85,B 0,C 180,E1 -26054.085,E2 -26054.085} C_VEL
LIN {X 0,Y 135.24,Z 524.37,A -85,B 0,C 180,E1 -26057.775,E2 -26057.775} C_VEL
LIN {X 0,Y 137.233,Z 513.852,A -85,B 0,C 180,E1 -26061.118,E2 -26061.118} C_VEL
LIN {X 0,Y 137.762,Z 508.698,A -85,B 0,C 180,E1 -26062.713,E2 -26062.713} C_VEL
LIN {X 0,Y 135.618,Z 499.649,A -85,B 0,C 180,E1 -26066.858,E2 -26066.858} C_VEL
LIN {X 0,Y 133.807,Z 493.076,A -85,B 0,C 180,E1 -26070.068,E2 -26070.068} C_VEL
LIN {X 0,Y 131.475,Z 486.48,A -85,B 0,C 180,E1 -26073.832,E2 -26073.832} C_VEL
LIN {X 0,Y 129.591,Z 481.803,A -85,B 0,C 180,E1 -26076.933,E2 -26076.933} C_VEL
LIN {X 0,Y 129.287,Z 480.581,A -85,B 0,C 180,E1 -26077.634,E2 -26077.634} C_VEL
LIN {X 0,Y 126.359,Z 474.895,A -85,B 0,C 180,E1 -26082.814,E2 -26082.814} C_VEL
LIN {X 0,Y 125.565,Z 472.15,A -85,B 0,C 180,E1 -26084.997,E2 -26084.997} C_VEL
LIN {X 0,Y 122.9,Z 467.265,A -85,B 0,C 180,E1 -26092.608,E2 -26092.608} C_VEL
LIN {X 0,Y 121.933,Z 464.749,A -85,B 0,C 180,E1 -26100,E2 -26100} C_VEL
LIN {X 0,Y 122.188,Z 466.692,A -85,B 0,C 180,E1 -26108.804,E2 -26108.804} C_VEL
LIN {X 0,Y 122.6,Z 467.994,A -85,B 0,C 180,E1 -26111.488,E2 -26111.488} C_VEL
LIN {X 0,Y 122.817,Z 470.405,A -85,B 0,C 180,E1 -26114.024,E2 -26114.024} C_VEL
LIN {X 0,Y 123.373,Z 478.324,A -85,B 0,C 180,E1 -26120.57,E2 -26120.57} C_VEL
LIN {X 0,Y 123.858,Z 479.847,A -85,B 0,C 180,E1 -26122.289,E2 -26122.289} C_VEL
LIN {X 0,Y 126.294,Z 485.022,A -85,B 0,C 180,E1 -26128.23,E2 -26128.23} C_VEL
LIN {X 0,Y 128.387,Z 490.384,A -85,B 0,C 180,E1 -26133.19,E2 -26133.19} C_VEL
LIN {X 0,Y 130.275,Z 496.023,A -85,B 0,C 180,E1 -26137.818,E2 -26137.818} C_VEL
LIN {X 0,Y 131.496,Z 501.129,A -85,B 0,C 180,E1 -26141.56,E2 -26141.56} C_VEL
LIN {X 0,Y 132.348,Z 506.861,A -85,B 0,C 180,E1 -26145.578,E2 -26145.578} C_VEL
LIN {X 0,Y 132.671,Z 512.112,A -85,B 0,C 180,E1 -26149.163,E2 -26149.163} C_VEL
LIN {X 0,Y 132.71,Z 514.052,A -85,B 0,C 180,E1 -26150.543,E2 -26150.543} C_VEL
LIN {X 0,Y 132.181,Z 515.548,A -85,B 0,C 180,E1 -26151.336,E2 -26151.336} C_VEL
LIN {X 0,Y 126.823,Z 523.669,A -85,B 0,C 180,E1 -26155.388,E2 -26155.388} C_VEL
LIN {X 0,Y 122.553,Z 529.625,A -85,B 0,C 180,E1 -26159.34,E2 -26159.34} C_VEL
LIN {X 0,Y 118.852,Z 534.564,A -85,B 0,C 180,E1 -26163.673,E2 -26163.673} C_VEL
LIN {X 0,Y 115.256,Z 538.8,A -85,B 0,C 180,E1 -26168.539,E2 -26168.539} C_VEL
LIN {X 0,Y 113.31,Z 541.031,A -85,B 0,C 180,E1 -26171.933,E2 -26171.933} C_VEL
LIN {X 0,Y 111.666,Z 542.85,A -85,B 0,C 180,E1 -26175.419,E2 -26175.419} C_VEL
LIN {X 0,Y 110.372,Z 544.216,A -85,B 0,C 180,E1 -26178.987,E2 -26178.987} C_VEL
LIN {X 0,Y 109.223,Z 545.733,A -85,B 0,C 180,E1 -26186.31,E2 -26186.31} C_VEL
LIN {X 0,Y 109.075,Z 545.95,A -85,B 0,C 180,E1 -26190,E2 -26190} C_VEL
LIN {X 0,Y 109.221,Z 545.761,A -85,B 0,C 180,E1 -26193.689,E2 -26193.689} C_VEL
LIN {X 0,Y 110.359,Z 544.28,A -85,B 0,C 180,E1 -26201.014,E2 -26201.014} C_VEL
LIN {X 0,Y 111.647,Z 542.944,A -85,B 0,C 180,E1 -26204.583,E2 -26204.583} C_VEL
LIN {X 0,Y 114.284,Z 540.114,A -85,B 0,C 180,E1 -26209.769,E2 -26209.769} C_VEL
LIN {X 0,Y 117.594,Z 536.289,A -85,B 0,C 180,E1 -26214.731,E2 -26214.731} C_VEL
LIN {X 0,Y 122.116,Z 530.352,A -85,B 0,C 180,E1 -26220.313,E2 -26220.313} C_VEL
LIN {X 0,Y 126.807,Z 523.957,A -85,B 0,C 180,E1 -26224.617,E2 -26224.617} C_VEL
LIN {X 0,Y 132.131,Z 515.903,A -85,B 0,C 180,E1 -26228.681,E2 -26228.681} C_VEL
LIN {X 0,Y 132.779,Z 514.417,A -85,B 0,C 180,E1 -26229.432,E2 -26229.432} C_VEL
LIN {X 0,Y 132.511,Z 507.282,A -85,B 0,C 180,E1 -26234.349,E2 -26234.349} C_VEL
LIN {X 0,Y 131.469,Z 500.548,A -85,B 0,C 180,E1 -26239.091,E2 -26239.091} C_VEL
LIN {X 0,Y 129.92,Z 494.755,A -85,B 0,C 180,E1 -26243.484,E2 -26243.484} C_VEL
LIN {X 0,Y 127.755,Z 488.465,A -85,B 0,C 180,E1 -26248.799,E2 -26248.799} C_VEL
LIN {X 0,Y 125.817,Z 483.699,A -85,B 0,C 180,E1 -26253.457,E2 -26253.457} C_VEL
LIN {X 0,Y 123.877,Z 479.642,A -85,B 0,C 180,E1 -26258.36,E2 -26258.36} C_VEL
LIN {X 0,Y 122.186,Z 476.592,A -85,B 0,C 180,E1 -26263.286,E2 -26263.286} C_VEL
LIN {X 0,Y 121.333,Z 474.992,A -85,B 0,C 180,E1 -26266.603,E2 -26266.603} C_VEL
LIN {X 0,Y 120.037,Z 472.689,A -85,B 0,C 180,E1 -26276.643,E2 -26276.643} C_VEL
LIN {X 0,Y 120.271,Z 472.347,A -85,B 0,C 180,E1 -26280.418,E2 -26280.418} C_VEL
LIN {X 0,Y 121.279,Z 474.546,A -85,B 0,C 180,E1 -26287.492,E2 -26287.492} C_VEL
LIN {X 0,Y 122.919,Z 478.181,A -85,B 0,C 180,E1 -26293.221,E2 -26293.221} C_VEL
LIN {X 0,Y 126.066,Z 486.848,A -85,B 0,C 180,E1 -26301.245,E2 -26301.245} C_VEL
LIN {X 0,Y 127.969,Z 492.398,A -85,B 0,C 180,E1 -26305.19,E2 -26305.19} C_VEL
LIN {X 0,Y 129.782,Z 499.146,A -85,B 0,C 180,E1 -26309.168,E2 -26309.168} C_VEL
LIN {X 0,Y 131.643,Z 507.508,A -85,B 0,C 180,E1 -26313.572,E2 -26313.572} C_VEL
LIN {X 0,Y 132.422,Z 512.861,A -85,B 0,C 180,E1 -26316.107,E2 -26316.107} C_VEL
LIN {X 0,Y 130.151,Z 523.604,A -85,B 0,C 180,E1 -26319.693,E2 -26319.693} C_VEL
LIN {X 0,Y 127.2,Z 533.729,A -85,B 0,C 180,E1 -26323.527,E2 -26323.527} C_VEL
LIN {X 0,Y 123.535,Z 543.541,A -85,B 0,C 180,E1 -26327.93,E2 -26327.93} C_VEL
LIN {X 0,Y 120.019,Z 551.134,A -85,B 0,C 180,E1 -26332.059,E2 -26332.059} C_VEL
LIN {X 0,Y 116.892,Z 557.332,A -85,B 0,C 180,E1 -26336.21,E2 -26336.21} C_VEL
LIN {X 0,Y 113.547,Z 562.375,A -85,B 0,C 180,E1 -26340.32,E2 -26340.32} C_VEL
LIN {X 0,Y 110.17,Z 567.293,A -85,B 0,C 180,E1 -26345.503,E2 -26345.503} C_VEL
LIN {X 0,Y 107.964,Z 571.135,A -85,B 0,C 180,E1 -26351.006,E2 -26351.006} C_VEL
LIN {X 0,Y 107.096,Z 573.158,A -85,B 0,C 180,E1 -26354.782,E2 -26354.782} C_VEL
LIN {X 0,Y 106.746,Z 575.51,A -85,B 0,C 180,E1 -26360.96,E2 -26360.96} C_VEL
LIN {X 0,Y 107.288,Z 576.655,A -85,B 0,C 180,E1 -26366.244,E2 -26366.244} C_VEL
LIN {X 0,Y 107.983,Z 576.994,A -85,B 0,C 180,E1 -26370,E2 -26370} C_VEL
LIN {X 0,Y 107.269,Z 576.636,A -85,B 0,C 180,E1 -26373.757,E2 -26373.757} C_VEL
LIN {X 0,Y 106.755,Z 574.691,A -85,B 0,C 180,E1 -26381.391,E2 -26381.391} C_VEL
LIN {X 0,Y 107.465,Z 572.126,A -85,B 0,C 180,E1 -26387.115,E2 -26387.115} C_VEL
LIN {X 0,Y 109.307,Z 568.592,A -85,B 0,C 180,E1 -26392.692,E2 -26392.692} C_VEL
LIN {X 0,Y 112.304,Z 564.018,A -85,B 0,C 180,E1 -26397.993,E2 -26397.993} C_VEL
LIN {X 0,Y 116.245,Z 558.263,A -85,B 0,C 180,E1 -26402.966,E2 -26402.966} C_VEL
LIN {X 0,Y 120.071,Z 550.966,A -85,B 0,C 180,E1 -26407.922,E2 -26407.922} C_VEL
LIN {X 0,Y 123.839,Z 542.528,A -85,B 0,C 180,E1 -26412.458,E2 -26412.458} C_VEL
LIN {X 0,Y 127.51,Z 532.471,A -85,B 0,C 180,E1 -26416.863,E2 -26416.863} C_VEL
LIN {X 0,Y 130.419,Z 521.985,A -85,B 0,C 180,E1 -26420.773,E2 -26420.773} C_VEL
LIN {X 0,Y 132.177,Z 513.434,A -85,B 0,C 180,E1 -26423.609,E2 -26423.609} C_VEL
LIN {X 0,Y 132.316,Z 511.684,A -85,B 0,C 180,E1 -26424.249,E2 -26424.249} C_VEL
LIN {X 0,Y 130.568,Z 502.76,A -85,B 0,C 180,E1 -26428.707,E2 -26428.707} C_VEL
LIN {X 0,Y 128.863,Z 496.164,A -85,B 0,C 180,E1 -26432.382,E2 -26432.382} C_VEL
LIN {X 0,Y 127.346,Z 491.14,A -85,B 0,C 180,E1 -26435.549,E2 -26435.549} C_VEL
LIN {X 0,Y 125.601,Z 485.796,A -85,B 0,C 180,E1 -26439.351,E2 -26439.351} C_VEL
LIN {X 0,Y 123.683,Z 481.451,A -85,B 0,C 180,E1 -26443.494,E2 -26443.494} C_VEL
LIN {X 0,Y 123.209,Z 479.479,A -85,B 0,C 180,E1 -26445.127,E2 -26445.127} C_VEL
LIN {X 0,Y 122.465,Z 477.622,A -85,B 0,C 180,E1 -26447.317,E2 -26447.317} C_VEL
LIN {X 0,Y 120.836,Z 473.964,A -85,B 0,C 180,E1 -26453.32,E2 -26453.32} C_VEL
LIN {X 0,Y 120.078,Z 471.72,A -85,B 0,C 180,E1 -26460,E2 -26460} C_VEL
LIN {X 0,Y 120.274,Z 473.861,A -85,B 0,C 180,E1 -26470.096,E2 -26470.096} C_VEL
LIN {X 0,Y 121.082,Z 474.721,A -85,B 0,C 180,E1 -26473.425,E2 -26473.425} C_VEL
LIN {X 0,Y 122.005,Z 476.147,A -85,B 0,C 180,E1 -26476.74,E2 -26476.74} C_VEL
LIN {X 0,Y 122.982,Z 478.45,A -85,B 0,C 180,E1 -26480.053,E2 -26480.053} C_VEL
LIN {X 0,Y 123.858,Z 479.847,A -85,B 0,C 180,E1 -26482.289,E2 -26482.289} C_VEL
LIN {X 0,Y 124.555,Z 482.373,A -85,B 0,C 180,E1 -26484.726,E2 -26484.726} C_VEL
LIN {X 0,Y 124.702,Z 485.751,A -85,B 0,C 180,E1 -26486.973,E2 -26486.973} C_VEL
LIN {X 0,Y 124.204,Z 495.672,A -85,B 0,C 180,E1 -26492.819,E2 -26492.819} C_VEL
LIN {X 0,Y 124.469,Z 497.725,A -85,B 0,C 180,E1 -26494.412,E2 -26494.412} C_VEL
LIN {X 0,Y 125.62,Z 502.44,A -85,B 0,C 180,E1 -26498.44,E2 -26498.44} C_VEL
LIN {X 0,Y 126.416,Z 508.227,A -85,B 0,C 180,E1 -26502.982,E2 -26502.982} C_VEL
LIN {X 0,Y 126.67,Z 514.2,A -85,B 0,C 180,E1 -26507.496,E2 -26507.496} C_VEL
LIN {X 0,Y 126.617,Z 516.585,A -85,B 0,C 180,E1 -26509.292,E2 -26509.292} C_VEL
LIN {X 0,Y 121.996,Z 523.472,A -85,B 0,C 180,E1 -26512.779,E2 -26512.779} C_VEL
LIN {X 0,Y 116.569,Z 530.625,A -85,B 0,C 180,E1 -26517.573,E2 -26517.573} C_VEL
LIN {X 0,Y 112.598,Z 535.57,A -85,B 0,C 180,E1 -26522.087,E2 -26522.087} C_VEL
LIN {X 0,Y 108.746,Z 539.806,A -85,B 0,C 180,E1 -26527.184,E2 -26527.184} C_VEL
LIN {X 0,Y 106.652,Z 542.037,A -85,B 0,C 180,E1 -26530.762,E2 -26530.762} C_VEL
LIN {X 0,Y 104.88,Z 543.856,A -85,B 0,C 180,E1 -26534.452,E2 -26534.452} C_VEL
LIN {X 0,Y 103.482,Z 545.221,A -85,B 0,C 180,E1 -26538.243,E2 -26538.243} C_VEL
LIN {X 0,Y 102.21,Z 546.738,A -85,B 0,C 180,E1 -26546.057,E2 -26546.057} C_VEL
LIN {X 0,Y 102.048,Z 546.955,A -85,B 0,C 180,E1 -26550,E2 -26550} C_VEL
LIN {X 0,Y 102.209,Z 546.766,A -85,B 0,C 180,E1 -26553.943,E2 -26553.943} C_VEL
LIN {X 0,Y 103.469,Z 545.284,A -85,B 0,C 180,E1 -26561.757,E2 -26561.757} C_VEL
LIN {X 0,Y 104.86,Z 543.948,A -85,B 0,C 180,E1 -26565.55,E2 -26565.55} C_VEL
LIN {X 0,Y 107.696,Z 541.119,A -85,B 0,C 180,E1 -26571.033,E2 -26571.033} C_VEL
LIN {X 0,Y 111.25,Z 537.293,A -85,B 0,C 180,E1 -26576.245,E2 -26576.245} C_VEL
LIN {X 0,Y 116.1,Z 531.359,A -85,B 0,C 180,E1 -26582.061,E2 -26582.061} C_VEL
LIN {X 0,Y 121.089,Z 524.96,A -85,B 0,C 180,E1 -26586.506,E2 -26586.506} C_VEL
LIN {X 0,Y 126.67,Z 516.915,A -85,B 0,C 180,E1 -26590.687,E2 -26590.687} C_VEL
LIN {X 0,Y 126.75,Z 511.098,A -85,B 0,C 180,E1 -26595.054,E2 -26595.054} C_VEL
LIN {X 0,Y 126.068,Z 504.527,A -85,B 0,C 180,E1 -26600.128,E2 -26600.128} C_VEL
LIN {X 0,Y 125.006,Z 499.559,A -85,B 0,C 180,E1 -26604.286,E2 -26604.286} C_VEL
LIN {X 0,Y 123.516,Z 494.198,A -85,B 0,C 180,E1 -26609.196,E2 -26609.196} C_VEL
LIN {X 0,Y 121.86,Z 489.313,A -85,B 0,C 180,E1 -26614.371,E2 -26614.371} C_VEL
LIN {X 0,Y 120.286,Z 485.504,A -85,B 0,C 180,E1 -26619.478,E2 -26619.478} C_VEL
LIN {X 0,Y 118.671,Z 481.806,A -85,B 0,C 180,E1 -26626.297,E2 -26626.297} C_VEL
LIN {X 0,Y 117.68,Z 480.063,A -85,B 0,C 180,E1 -26633.14,E2 -26633.14} C_VEL
LIN {X 0,Y 118.016,Z 479.025,A -85,B 0,C 180,E1 -26640,E2 -26640} C_VEL
LIN {X 0,Y 118.838,Z 481.052,A -85,B 0,C 180,E1 -26646.793,E2 -26646.793} C_VEL
LIN {X 0,Y 120.124,Z 484.497,A -85,B 0,C 180,E1 -26652.413,E2 -26652.413} C_VEL
LIN {X 0,Y 122.461,Z 492.521,A -85,B 0,C 180,E1 -26660.141,E2 -26660.141} C_VEL
LIN {X 0,Y 123.953,Z 498.061,A -85,B 0,C 180,E1 -26664.274,E2 -26664.274} C_VEL
LIN {X 0,Y 125.375,Z 504.67,A -85,B 0,C 180,E1 -26668.455,E2 -26668.455} C_VEL
LIN {X 0,Y 126.697,Z 512.969,A -85,B 0,C 180,E1 -26673.094,E2 -26673.094} C_VEL
LIN {X 0,Y 126.911,Z 515.922,A -85,B 0,C 180,E1 -26674.582,E2 -26674.582} C_VEL
LIN {X 0,Y 123.94,Z 526.921,A -85,B 0,C 180,E1 -26678.591,E2 -26678.591} C_VEL
LIN {X 0,Y 120.905,Z 535.55,A -85,B 0,C 180,E1 -26682.172,E2 -26682.172} C_VEL
LIN {X 0,Y 116.912,Z 544.925,A -85,B 0,C 180,E1 -26686.794,E2 -26686.794} C_VEL
LIN {X 0,Y 112.892,Z 552.695,A -85,B 0,C 180,E1 -26691.498,E2 -26691.498} C_VEL
LIN {X 0,Y 110.228,Z 557.369,A -85,B 0,C 180,E1 -26694.983,E2 -26694.983} C_VEL
LIN {X 0,Y 106.067,Z 563.116,A -85,B 0,C 180,E1 -26700.202,E2 -26700.202} C_VEL
LIN {X 0,Y 102.74,Z 567.656,A -85,B 0,C 180,E1 -26705.768,E2 -26705.768} C_VEL
LIN {X 0,Y 100.65,Z 571.162,A -85,B 0,C 180,E1 -26711.687,E2 -26711.687} C_VEL
LIN {X 0,Y 99.734,Z 573.701,A -85,B 0,C 180,E1 -26717.796,E2 -26717.796} C_VEL
LIN {X 0,Y 100.165,Z 575.634,A -85,B 0,C 180,E1 -26725.977,E2 -26725.977} C_VEL
LIN {X 0,Y 100.886,Z 575.979,A -85,B 0,C 180,E1 -26730,E2 -26730} C_VEL
LIN {X 0,Y 100.15,Z 575.615,A -85,B 0,C 180,E1 -26734.024,E2 -26734.024} C_VEL
LIN {X 0,Y 99.693,Z 574.563,A -85,B 0,C 180,E1 -26739.265,E2 -26739.265} C_VEL
LIN {X 0,Y 100.193,Z 572.079,A -85,B 0,C 180,E1 -26746.295,E2 -26746.295} C_VEL
LIN {X 0,Y 101.9,Z 568.88,A -85,B 0,C 180,E1 -26752.293,E2 -26752.293} C_VEL
LIN {X 0,Y 104.774,Z 564.658,A -85,B 0,C 180,E1 -26758.005,E2 -26758.005} C_VEL
LIN {X 0,Y 109.482,Z 558.392,A -85,B 0,C 180,E1 -26764.062,E2 -26764.062} C_VEL
LIN {X 0,Y 113.608,Z 551.214,A -85,B 0,C 180,E1 -26769.353,E2 -26769.353} C_VEL
LIN {X 0,Y 116.871,Z 544.738,A -85,B 0,C 180,E1 -26773.197,E2 -26773.197} C_VEL
LIN {X 0,Y 120.939,Z 535.29,A -85,B 0,C 180,E1 -26777.811,E2 -26777.811} C_VEL
LIN {X 0,Y 124.518,Z 524.6,A -85,B 0,C 180,E1 -26782.204,E2 -26782.204} C_VEL
LIN {X 0,Y 126.775,Z 515.767,A -85,B 0,C 180,E1 -26785.375,E2 -26785.375} C_VEL
LIN {X 0,Y 126.395,Z 511.493,A -85,B 0,C 180,E1 -26787.55,E2 -26787.55} C_VEL
LIN {X 0,Y 124.996,Z 502.998,A -85,B 0,C 180,E1 -26792.363,E2 -26792.363} C_VEL
LIN {X 0,Y 123.482,Z 496.691,A -85,B 0,C 180,E1 -26796.521,E2 -26796.521} C_VEL
LIN {X 0,Y 122.305,Z 492.22,A -85,B 0,C 180,E1 -26799.832,E2 -26799.832} C_VEL
LIN {X 0,Y 120.174,Z 485.244,A -85,B 0,C 180,E1 -26806.472,E2 -26806.472} C_VEL
LIN {X 0,Y 118.885,Z 481.823,A -85,B 0,C 180,E1 -26811.501,E2 -26811.501} C_VEL
LIN {X 0,Y 118.604,Z 480.813,A -85,B 0,C 180,E1 -26813.194,E2 -26813.194} C_VEL
LIN {X 0,Y 117.839,Z 478.588,A -85,B 0,C 180,E1 -26820,E2 -26820} C_VEL
LIN {X 0,Y 117.467,Z 479.869,A -85,B 0,C 180,E1 -26827.27,E2 -26827.27} C_VEL
LIN {X 0,Y 118.469,Z 481.474,A -85,B 0,C 180,E1 -26833.727,E2 -26833.727} C_VEL
LIN {X 0,Y 120.074,Z 485.229,A -85,B 0,C 180,E1 -26840.56,E2 -26840.56} C_VEL
LIN {X 0,Y 121.079,Z 487.778,A -85,B 0,C 180,E1 -26843.974,E2 -26843.974} C_VEL
LIN {X 0,Y 122.238,Z 490.539,A -85,B 0,C 180,E1 -26847.385,E2 -26847.385} C_VEL
LIN {X 0,Y 123.909,Z 495.745,A -85,B 0,C 180,E1 -26852.602,E2 -26852.602} C_VEL
LIN {X 0,Y 124.469,Z 497.725,A -85,B 0,C 180,E1 -26854.412,E2 -26854.412} C_VEL
LIN {X 0,Y 124.694,Z 499.785,A -85,B 0,C 180,E1 -26855.968,E2 -26855.968} C_VEL
LIN {X 0,Y 124.265,Z 503.446,A -85,B 0,C 180,E1 -26858.135,E2 -26858.135} C_VEL
LIN {X 0,Y 123.226,Z 507.364,A -85,B 0,C 180,E1 -26860.2,E2 -26860.2} C_VEL
LIN {X 0,Y 121.011,Z 514.802,A -85,B 0,C 180,E1 -26864.54,E2 -26864.54} C_VEL
LIN {X 0,Y 120.689,Z 516.914,A -85,B 0,C 180,E1 -26866.139,E2 -26866.139} C_VEL
LIN {X 0,Y 120.491,Z 519.019,A -85,B 0,C 180,E1 -26867.873,E2 -26867.873} C_VEL
LIN {X 0,Y 114.583,Z 526.889,A -85,B 0,C 180,E1 -26872.167,E2 -26872.167} C_VEL
LIN {X 0,Y 109.612,Z 533.027,A -85,B 0,C 180,E1 -26876.828,E2 -26876.828} C_VEL
LIN {X 0,Y 105.041,Z 538.125,A -85,B 0,C 180,E1 -26882.072,E2 -26882.072} C_VEL
LIN {X 0,Y 101.184,Z 541.998,A -85,B 0,C 180,E1 -26887.541,E2 -26887.541} C_VEL
LIN {X 0,Y 98.127,Z 544.862,A -85,B 0,C 180,E1 -26893.352,E2 -26893.352} C_VEL
LIN {X 0,Y 96.612,Z 546.227,A -85,B 0,C 180,E1 -26897.394,E2 -26897.394} C_VEL
LIN {X 0,Y 95.2,Z 547.744,A -85,B 0,C 180,E1 -26905.766,E2 -26905.766} C_VEL
LIN {X 0,Y 95.02,Z 547.96,A -85,B 0,C 180,E1 -26910,E2 -26910} C_VEL
LIN {X 0,Y 95.199,Z 547.771,A -85,B 0,C 180,E1 -26914.233,E2 -26914.233} C_VEL
LIN {X 0,Y 96.599,Z 546.289,A -85,B 0,C 180,E1 -26922.607,E2 -26922.607} C_VEL
LIN {X 0,Y 98.107,Z 544.953,A -85,B 0,C 180,E1 -26926.651,E2 -26926.651} C_VEL
LIN {X 0,Y 101.168,Z 542.123,A -85,B 0,C 180,E1 -26932.462,E2 -26932.462} C_VEL
LIN {X 0,Y 104.992,Z 538.297,A -85,B 0,C 180,E1 -26937.941,E2 -26937.941} C_VEL
LIN {X 0,Y 110.214,Z 532.355,A -85,B 0,C 180,E1 -26944.007,E2 -26944.007} C_VEL
LIN {X 0,Y 115.516,Z 525.963,A -85,B 0,C 180,E1 -26948.58,E2 -26948.58} C_VEL
LIN {X 0,Y 120.457,Z 519.361,A -85,B 0,C 180,E1 -26952.141,E2 -26952.141} C_VEL
LIN {X 0,Y 120.91,Z 514.882,A -85,B 0,C 180,E1 -26955.772,E2 -26955.772} C_VEL
LIN {X 0,Y 120.728,Z 509.657,A -85,B 0,C 180,E1 -26960.182,E2 -26960.182} C_VEL
LIN {X 0,Y 119.978,Z 504.268,A -85,B 0,C 180,E1 -26965.093,E2 -26965.093} C_VEL
LIN {X 0,Y 118.978,Z 499.494,A -85,B 0,C 180,E1 -26969.861,E2 -26969.861} C_VEL
LIN {X 0,Y 117.736,Z 494.782,A -85,B 0,C 180,E1 -26975.301,E2 -26975.301} C_VEL
LIN {X 0,Y 116.954,Z 492.222,A -85,B 0,C 180,E1 -26978.866,E2 -26978.866} C_VEL
LIN {X 0,Y 115.544,Z 488.133,A -85,B 0,C 180,E1 -26986.706,E2 -26986.706} C_VEL
LIN {X 0,Y 114.969,Z 486.022,A -85,B 0,C 180,E1 -26996.495,E2 -26996.495} C_VEL
LIN {X 0,Y 115.352,Z 485.669,A -85,B 0,C 180,E1 -27000,E2 -27000} C_VEL
LIN {X 0,Y 116.096,Z 487.914,A -85,B 0,C 180,E1 -27006.954,E2 -27006.954} C_VEL
LIN {X 0,Y 116.71,Z 489.935,A -85,B 0,C 180,E1 -27010.408,E2 -27010.408} C_VEL
LIN {X 0,Y 117.048,Z 491.239,A -85,B 0,C 180,E1 -27012.131,E2 -27012.131} C_VEL
LIN {X 0,Y 118.617,Z 498.019,A -85,B 0,C 180,E1 -27019.016,E2 -27019.016} C_VEL
LIN {X 0,Y 119.701,Z 503.512,A -85,B 0,C 180,E1 -27023.348,E2 -27023.348} C_VEL
LIN {X 0,Y 120.707,Z 510.036,A -85,B 0,C 180,E1 -27027.761,E2 -27027.761} C_VEL
LIN {X 0,Y 121.43,Z 517.262,A -85,B 0,C 180,E1 -27032.114,E2 -27032.114} C_VEL
LIN {X 0,Y 121.438,Z 518.625,A -85,B 0,C 180,E1 -27032.839,E2 -27032.839} C_VEL
LIN {X 0,Y 118.048,Z 529.031,A -85,B 0,C 180,E1 -27036.962,E2 -27036.962} C_VEL
LIN {X 0,Y 114.283,Z 538.141,A -85,B 0,C 180,E1 -27041.12,E2 -27041.12} C_VEL
LIN {X 0,Y 110.342,Z 546.194,A -85,B 0,C 180,E1 -27045.523,E2 -27045.523} C_VEL
LIN {X 0,Y 105.742,Z 554.058,A -85,B 0,C 180,E1 -27050.846,E2 -27050.846} C_VEL
LIN {X 0,Y 102.752,Z 558.633,A -85,B 0,C 180,E1 -27054.693,E2 -27054.693} C_VEL
LIN {X 0,Y 98.544,Z 563.746,A -85,B 0,C 180,E1 -27060.051,E2 -27060.051} C_VEL
LIN {X 0,Y 95.302,Z 567.931,A -85,B 0,C 180,E1 -27066.072,E2 -27066.072} C_VEL
LIN {X 0,Y 93.353,Z 571.111,A -85,B 0,C 180,E1 -27072.475,E2 -27072.475} C_VEL
LIN {X 0,Y 92.673,Z 573.845,A -85,B 0,C 180,E1 -27081.276,E2 -27081.276} C_VEL
LIN {X 0,Y 93.049,Z 574.614,A -85,B 0,C 180,E1 -27085.669,E2 -27085.669} C_VEL
LIN {X 0,Y 93.785,Z 574.964,A -85,B 0,C 180,E1 -27090,E2 -27090} C_VEL
LIN {X 0,Y 93.037,Z 574.595,A -85,B 0,C 180,E1 -27094.333,E2 -27094.333} C_VEL
LIN {X 0,Y 92.633,Z 573.645,A -85,B 0,C 180,E1 -27099.495,E2 -27099.495} C_VEL
LIN {X 0,Y 93.351,Z 571.056,A -85,B 0,C 180,E1 -27107.527,E2 -27107.527} C_VEL
LIN {X 0,Y 95.286,Z 567.851,A -85,B 0,C 180,E1 -27113.933,E2 -27113.933} C_VEL
LIN {X 0,Y 98.528,Z 563.636,A -85,B 0,C 180,E1 -27119.955,E2 -27119.955} C_VEL
LIN {X 0,Y 102.903,Z 558.302,A -85,B 0,C 180,E1 -27125.488,E2 -27125.488} C_VEL
LIN {X 0,Y 107.235,Z 551.462,A -85,B 0,C 180,E1 -27130.95,E2 -27130.95} C_VEL
LIN {X 0,Y 111.087,Z 544.477,A -85,B 0,C 180,E1 -27135.394,E2 -27135.394} C_VEL
LIN {X 0,Y 115.107,Z 536.089,A -85,B 0,C 180,E1 -27139.748,E2 -27139.748} C_VEL
LIN {X 0,Y 118.891,Z 526.201,A -85,B 0,C 180,E1 -27144.098,E2 -27144.098} C_VEL
LIN {X 0,Y 121.335,Z 518.381,A -85,B 0,C 180,E1 -27147.147,E2 -27147.147} C_VEL
LIN {X 0,Y 120.761,Z 511.44,A -85,B 0,C 180,E1 -27151.212,E2 -27151.212} C_VEL
LIN {X 0,Y 119.855,Z 505.214,A -85,B 0,C 180,E1 -27155.286,E2 -27155.286} C_VEL
LIN {X 0,Y 118.842,Z 500.006,A -85,B 0,C 180,E1 -27159.217,E2 -27159.217} C_VEL
LIN {X 0,Y 118.478,Z 497.715,A -85,B 0,C 180,E1 -27160.96,E2 -27160.96} C_VEL
LIN {X 0,Y 116.871,Z 490.941,A -85,B 0,C 180,E1 -27167.85,E2 -27167.85} C_VEL
LIN {X 0,Y 115.886,Z 487.667,A -85,B 0,C 180,E1 -27173.033,E2 -27173.033} C_VEL
LIN {X 0,Y 115.205,Z 485.247,A -85,B 0,C 180,E1 -27180,E2 -27180} C_VEL
LIN {X 0,Y 114.681,Z 486.428,A -85,B 0,C 180,E1 -27187.283,E2 -27187.283} C_VEL
LIN {X 0,Y 115.436,Z 488.186,A -85,B 0,C 180,E1 -27194.095,E2 -27194.095} C_VEL
LIN {X 0,Y 116.766,Z 491.937,A -85,B 0,C 180,E1 -27201.17,E2 -27201.17} C_VEL
LIN {X 0,Y 118.058,Z 496.125,A -85,B 0,C 180,E1 -27206.752,E2 -27206.752} C_VEL
LIN {X 0,Y 119.233,Z 501.007,A -85,B 0,C 180,E1 -27212.039,E2 -27212.039} C_VEL
LIN {X 0,Y 120.299,Z 506.444,A -85,B 0,C 180,E1 -27217.275,E2 -27217.275} C_VEL
LIN {X 0,Y 120.753,Z 511.938,A -85,B 0,C 180,E1 -27222.013,E2 -27222.013} C_VEL
LIN {X 0,Y 120.689,Z 516.914,A -85,B 0,C 180,E1 -27226.139,E2 -27226.139} C_VEL
LIN {X 0,Y 119.849,Z 518.792,A -85,B 0,C 180,E1 -27227.268,E2 -27227.268} C_VEL
LIN {X 0,Y 117.593,Z 521.338,A -85,B 0,C 180,E1 -27228.225,E2 -27228.225} C_VEL
LIN {X 0,Y 109.88,Z 527.594,A -85,B 0,C 180,E1 -27230.042,E2 -27230.042} C_VEL
LIN {X 0,Y 107.375,Z 529.937,A -85,B 0,C 180,E1 -27231.341,E2 -27231.341} C_VEL
LIN {X 0,Y 101.967,Z 535.934,A -85,B 0,C 180,E1 -27236.537,E2 -27236.537} C_VEL
LIN {X 0,Y 97.371,Z 540.526,A -85,B 0,C 180,E1 -27242.02,E2 -27242.02} C_VEL
LIN {X 0,Y 93.496,Z 544.049,A -85,B 0,C 180,E1 -27247.923,E2 -27247.923} C_VEL
LIN {X 0,Y 91.416,Z 545.868,A -85,B 0,C 180,E1 -27252.09,E2 -27252.09} C_VEL
LIN {X 0,Y 89.766,Z 547.233,A -85,B 0,C 180,E1 -27256.415,E2 -27256.415} C_VEL
LIN {X 0,Y 88.193,Z 548.749,A -85,B 0,C 180,E1 -27265.429,E2 -27265.429} C_VEL
LIN {X 0,Y 87.992,Z 548.965,A -85,B 0,C 180,E1 -27270,E2 -27270} C_VEL
LIN {X 0,Y 88.192,Z 548.776,A -85,B 0,C 180,E1 -27274.57,E2 -27274.57} C_VEL
LIN {X 0,Y 89.754,Z 547.294,A -85,B 0,C 180,E1 -27283.586,E2 -27283.586} C_VEL
LIN {X 0,Y 91.396,Z 545.957,A -85,B 0,C 180,E1 -27287.913,E2 -27287.913} C_VEL
LIN {X 0,Y 94.712,Z 543.127,A -85,B 0,C 180,E1 -27294.087,E2 -27294.087} C_VEL
LIN {X 0,Y 98.838,Z 539.301,A -85,B 0,C 180,E1 -27299.851,E2 -27299.851} C_VEL
LIN {X 0,Y 104.463,Z 533.358,A -85,B 0,C 180,E1 -27306.164,E2 -27306.164} C_VEL
LIN {X 0,Y 110.109,Z 526.967,A -85,B 0,C 180,E1 -27310.861,E2 -27310.861} C_VEL
LIN {X 0,Y 114.266,Z 521.816,A -85,B 0,C 180,E1 -27313.784,E2 -27313.784} C_VEL
LIN {X 0,Y 114.76,Z 520.481,A -85,B 0,C 180,E1 -27314.77,E2 -27314.77} C_VEL
LIN {X 0,Y 115.134,Z 516.221,A -85,B 0,C 180,E1 -27318.685,E2 -27318.685} C_VEL
LIN {X 0,Y 115.127,Z 512.195,A -85,B 0,C 180,E1 -27322.523,E2 -27322.523} C_VEL
LIN {X 0,Y 114.756,Z 508.254,A -85,B 0,C 180,E1 -27326.551,E2 -27326.551} C_VEL
LIN {X 0,Y 114.062,Z 503.369,A -85,B 0,C 180,E1 -27332.009,E2 -27332.009} C_VEL
LIN {X 0,Y 113.433,Z 500.123,A -85,B 0,C 180,E1 -27336.251,E2 -27336.251} C_VEL
LIN {X 0,Y 112.579,Z 496.799,A -85,B 0,C 180,E1 -27341.812,E2 -27341.812} C_VEL
LIN {X 0,Y 112.207,Z 495.048,A -85,B 0,C 180,E1 -27345.49,E2 -27345.49} C_VEL
LIN {X 0,Y 111.89,Z 493.787,A -85,B 0,C 180,E1 -27349.138,E2 -27349.138} C_VEL
LIN {X 0,Y 111.89,Z 492.477,A -85,B 0,C 180,E1 -27356.399,E2 -27356.399} C_VEL
LIN {X 0,Y 112.326,Z 492.155,A -85,B 0,C 180,E1 -27360,E2 -27360} C_VEL
LIN {X 0,Y 112.995,Z 494.575,A -85,B 0,C 180,E1 -27367.146,E2 -27367.146} C_VEL
LIN {X 0,Y 113.492,Z 496.781,A -85,B 0,C 180,E1 -27370.706,E2 -27370.706} C_VEL
LIN {X 0,Y 114.541,Z 503.35,A -85,B 0,C 180,E1 -27377.866,E2 -27377.866} C_VEL
LIN {X 0,Y 115.252,Z 509.301,A -85,B 0,C 180,E1 -27382.794,E2 -27382.794} C_VEL
LIN {X 0,Y 115.78,Z 515.229,A -85,B 0,C 180,E1 -27387.081,E2 -27387.081} C_VEL
LIN {X 0,Y 115.972,Z 521.004,A -85,B 0,C 180,E1 -27390.844,E2 -27390.844} C_VEL
LIN {X 0,Y 112.812,Z 529.572,A -85,B 0,C 180,E1 -27394.534,E2 -27394.534} C_VEL
LIN {X 0,Y 108.52,Z 538.789,A -85,B 0,C 180,E1 -27399,E2 -27399} C_VEL
LIN {X 0,Y 104.283,Z 546.57,A -85,B 0,C 180,E1 -27403.575,E2 -27403.575} C_VEL
LIN {X 0,Y 99.365,Z 554.191,A -85,B 0,C 180,E1 -27409.138,E2 -27409.138} C_VEL
LIN {X 0,Y 97.096,Z 557.407,A -85,B 0,C 180,E1 -27412.031,E2 -27412.031} C_VEL
LIN {X 0,Y 92.424,Z 562.725,A -85,B 0,C 180,E1 -27417.84,E2 -27417.84} C_VEL
LIN {X 0,Y 88.79,Z 566.906,A -85,B 0,C 180,E1 -27424.193,E2 -27424.193} C_VEL
LIN {X 0,Y 86.532,Z 570.085,A -85,B 0,C 180,E1 -27431.042,E2 -27431.042} C_VEL
LIN {X 0,Y 85.606,Z 572.822,A -85,B 0,C 180,E1 -27440.55,E2 -27440.55} C_VEL
LIN {X 0,Y 85.942,Z 573.594,A -85,B 0,C 180,E1 -27445.31,E2 -27445.31} C_VEL
LIN {X 0,Y 86.678,Z 573.947,A -85,B 0,C 180,E1 -27450,E2 -27450} C_VEL
LIN {X 0,Y 85.933,Z 573.576,A -85,B 0,C 180,E1 -27454.692,E2 -27454.692} C_VEL
LIN {X 0,Y 85.586,Z 572.72,A -85,B 0,C 180,E1 -27459.803,E2 -27459.803} C_VEL
LIN {X 0,Y 86.529,Z 570.028,A -85,B 0,C 180,E1 -27468.959,E2 -27468.959} C_VEL
LIN {X 0,Y 88.773,Z 566.823,A -85,B 0,C 180,E1 -27475.813,E2 -27475.813} C_VEL
LIN {X 0,Y 93.376,Z 561.552,A -85,B 0,C 180,E1 -27483.439,E2 -27483.439} C_VEL
LIN {X 0,Y 97.849,Z 556.202,A -85,B 0,C 180,E1 -27488.938,E2 -27488.938} C_VEL
LIN {X 0,Y 102.554,Z 549.085,A -85,B 0,C 180,E1 -27494.623,E2 -27494.623} C_VEL
LIN {X 0,Y 107.11,Z 541.2,A -85,B 0,C 180,E1 -27499.56,E2 -27499.56} C_VEL
LIN {X 0,Y 111.11,Z 533.064,A -85,B 0,C 180,E1 -27503.753,E2 -27503.753} C_VEL
LIN {X 0,Y 114.758,Z 524.147,A -85,B 0,C 180,E1 -27507.701,E2 -27507.701} C_VEL
LIN {X 0,Y 115.872,Z 520.468,A -85,B 0,C 180,E1 -27509.32,E2 -27509.32} C_VEL
LIN {X 0,Y 115.491,Z 512.242,A -85,B 0,C 180,E1 -27514.788,E2 -27514.788} C_VEL
LIN {X 0,Y 114.789,Z 506.289,A -85,B 0,C 180,E1 -27519.388,E2 -27519.388} C_VEL
LIN {X 0,Y 114.178,Z 502.224,A -85,B 0,C 180,E1 -27523.019,E2 -27523.019} C_VEL
LIN {X 0,Y 113.329,Z 496.487,A -85,B 0,C 180,E1 -27529.278,E2 -27529.278} C_VEL
LIN {X 0,Y 112.793,Z 494.344,A -85,B 0,C 180,E1 -27532.841,E2 -27532.841} C_VEL
LIN {X 0,Y 112.202,Z 491.744,A -85,B 0,C 180,E1 -27540,E2 -27540} C_VEL
LIN {X 0,Y 111.536,Z 492.81,A -85,B 0,C 180,E1 -27547.267,E2 -27547.267} C_VEL
LIN {X 0,Y 111.687,Z 493.54,A -85,B 0,C 180,E1 -27550.882,E2 -27550.882} C_VEL
LIN {X 0,Y 112.038,Z 494.734,A -85,B 0,C 180,E1 -27554.532,E2 -27554.532} C_VEL
LIN {X 0,Y 112.865,Z 497.969,A -85,B 0,C 180,E1 -27560.926,E2 -27560.926} C_VEL
LIN {X 0,Y 113.573,Z 501.236,A -85,B 0,C 180,E1 -27565.669,E2 -27565.669} C_VEL
LIN {X 0,Y 114.385,Z 506.111,A -85,B 0,C 180,E1 -27571.482,E2 -27571.482} C_VEL
LIN {X 0,Y 114.957,Z 510.685,A -85,B 0,C 180,E1 -27576.337,E2 -27576.337} C_VEL
LIN {X 0,Y 115.026,Z 515.883,A -85,B 0,C 180,E1 -27581.248,E2 -27581.248} C_VEL
LIN {X 0,Y 114.693,Z 520.164,A -85,B 0,C 180,E1 -27585.195,E2 -27585.195} C_VEL
LIN {X 0,Y 114.278,Z 521.486,A -85,B 0,C 180,E1 -27586.221,E2 -27586.221} C_VEL
LIN {X 0,Y 108.149,Z 529.042,A -85,B 0,C 180,E1 -27590.683,E2 -27590.683} C_VEL
LIN {X 0,Y 107.375,Z 529.937,A -85,B 0,C 180,E1 -27591.341,E2 -27591.341} C_VEL
LIN {X 0,Y 104.214,Z 533.027,A -85,B 0,C 180,E1 -27593.488,E2 -27593.488} C_VEL
LIN {X 0,Y 97.669,Z 537.758,A -85,B 0,C 180,E1 -27596.793,E2 -27596.793} C_VEL
LIN {X 0,Y 91.288,Z 541.849,A -85,B 0,C 180,E1 -27600.702,E2 -27600.702} C_VEL
LIN {X 0,Y 88.532,Z 543.849,A -85,B 0,C 180,E1 -27603.767,E2 -27603.767} C_VEL
LIN {X 0,Y 84.756,Z 546.873,A -85,B 0,C 180,E1 -27610.629,E2 -27610.629} C_VEL
LIN {X 0,Y 82.951,Z 548.238,A -85,B 0,C 180,E1 -27615.275,E2 -27615.275} C_VEL
LIN {X 0,Y 81.189,Z 549.754,A -85,B 0,C 180,E1 -27625.034,E2 -27625.034} C_VEL
LIN {X 0,Y 80.965,Z 549.971,A -85,B 0,C 180,E1 -27630,E2 -27630} C_VEL
LIN {X 0,Y 81.188,Z 549.781,A -85,B 0,C 180,E1 -27634.966,E2 -27634.966} C_VEL
LIN {X 0,Y 82.939,Z 548.299,A -85,B 0,C 180,E1 -27644.727,E2 -27644.727} C_VEL
LIN {X 0,Y 84.736,Z 546.962,A -85,B 0,C 180,E1 -27649.375,E2 -27649.375} C_VEL
LIN {X 0,Y 88.342,Z 544.131,A -85,B 0,C 180,E1 -27655.947,E2 -27655.947} C_VEL
LIN {X 0,Y 92.809,Z 540.305,A -85,B 0,C 180,E1 -27662.011,E2 -27662.011} C_VEL
LIN {X 0,Y 98.872,Z 534.365,A -85,B 0,C 180,E1 -27668.564,E2 -27668.564} C_VEL
LIN {X 0,Y 104.895,Z 527.97,A -85,B 0,C 180,E1 -27673.374,E2 -27673.374} C_VEL
LIN {X 0,Y 108.157,Z 524.162,A -85,B 0,C 180,E1 -27675.625,E2 -27675.625} C_VEL
LIN {X 0,Y 108.863,Z 523.099,A -85,B 0,C 180,E1 -27676.355,E2 -27676.355} C_VEL
LIN {X 0,Y 109.427,Z 519.1,A -85,B 0,C 180,E1 -27680.417,E2 -27680.417} C_VEL
LIN {X 0,Y 109.605,Z 515.049,A -85,B 0,C 180,E1 -27684.753,E2 -27684.753} C_VEL
LIN {X 0,Y 109.364,Z 509.666,A -85,B 0,C 180,E1 -27691.186,E2 -27691.186} C_VEL
LIN {X 0,Y 108.971,Z 505.306,A -85,B 0,C 180,E1 -27697.234,E2 -27697.234} C_VEL
LIN {X 0,Y 108.628,Z 503.155,A -85,B 0,C 180,E1 -27701.126,E2 -27701.126} C_VEL
LIN {X 0,Y 108.324,Z 500.731,A -85,B 0,C 180,E1 -27706.702,E2 -27706.702} C_VEL
LIN {X 0,Y 108.192,Z 499.281,A -85,B 0,C 180,E1 -27712.535,E2 -27712.535} C_VEL
LIN {X 0,Y 108.951,Z 498.468,A -85,B 0,C 180,E1 -27720,E2 -27720} C_VEL
LIN {X 0,Y 109.129,Z 499.557,A -85,B 0,C 180,E1 -27723.692,E2 -27723.692} C_VEL
LIN {X 0,Y 109.529,Z 501.058,A -85,B 0,C 180,E1 -27727.373,E2 -27727.373} C_VEL
LIN {X 0,Y 109.688,Z 502.163,A -85,B 0,C 180,E1 -27729.217,E2 -27729.217} C_VEL
LIN {X 0,Y 110.24,Z 508.871,A -85,B 0,C 180,E1 -27737.005,E2 -27737.005} C_VEL
LIN {X 0,Y 110.57,Z 514.998,A -85,B 0,C 180,E1 -27742.418,E2 -27742.418} C_VEL
LIN {X 0,Y 110.579,Z 521.248,A -85,B 0,C 180,E1 -27747.154,E2 -27747.154} C_VEL
LIN {X 0,Y 110.502,Z 523.113,A -85,B 0,C 180,E1 -27748.488,E2 -27748.488} C_VEL
LIN {X 0,Y 110.21,Z 524.633,A -85,B 0,C 180,E1 -27749.383,E2 -27749.383} C_VEL
LIN {X 0,Y 105.801,Z 534.163,A -85,B 0,C 180,E1 -27753.867,E2 -27753.867} C_VEL
LIN {X 0,Y 100.685,Z 543.191,A -85,B 0,C 180,E1 -27758.918,E2 -27758.918} C_VEL
LIN {X 0,Y 96.522,Z 549.528,A -85,B 0,C 180,E1 -27763.271,E2 -27763.271} C_VEL
LIN {X 0,Y 91.496,Z 556.372,A -85,B 0,C 180,E1 -27769.239,E2 -27769.239} C_VEL
LIN {X 0,Y 86.465,Z 561.705,A -85,B 0,C 180,E1 -27775.322,E2 -27775.322} C_VEL
LIN {X 0,Y 82.401,Z 565.882,A -85,B 0,C 180,E1 -27782.025,E2 -27782.025} C_VEL
LIN {X 0,Y 79.785,Z 569.06,A -85,B 0,C 180,E1 -27789.369,E2 -27789.369} C_VEL
LIN {X 0,Y 78.56,Z 571.812,A -85,B 0,C 180,E1 -27799.758,E2 -27799.758} C_VEL
LIN {X 0,Y 78.84,Z 572.575,A -85,B 0,C 180,E1 -27804.886,E2 -27804.886} C_VEL
LIN {X 0,Y 79.569,Z 572.93,A -85,B 0,C 180,E1 -27810,E2 -27810} C_VEL
LIN {X 0,Y 78.829,Z 572.556,A -85,B 0,C 180,E1 -27815.115,E2 -27815.115} C_VEL
LIN {X 0,Y 78.843,Z 570.587,A -85,B 0,C 180,E1 -27825.511,E2 -27825.511} C_VEL
LIN {X 0,Y 80.475,Z 568.018,A -85,B 0,C 180,E1 -27833.141,E2 -27833.141} C_VEL
LIN {X 0,Y 83.593,Z 564.488,A -85,B 0,C 180,E1 -27840.295,E2 -27840.295} C_VEL
LIN {X 0,Y 88.879,Z 559.101,A -85,B 0,C 180,E1 -27847.746,E2 -27847.746} C_VEL
LIN {X 0,Y 92.244,Z 555.148,A -85,B 0,C 180,E1 -27851.81,E2 -27851.81} C_VEL
LIN {X 0,Y 97.407,Z 548.021,A -85,B 0,C 180,E1 -27857.693,E2 -27857.693} C_VEL
LIN {X 0,Y 102.94,Z 539.136,A -85,B 0,C 180,E1 -27863.359,E2 -27863.359} C_VEL
LIN {X 0,Y 107.645,Z 529.997,A -85,B 0,C 180,E1 -27868.077,E2 -27868.077} C_VEL
LIN {X 0,Y 110.103,Z 524.455,A -85,B 0,C 180,E1 -27870.572,E2 -27870.572} C_VEL
LIN {X 0,Y 110.449,Z 521.449,A -85,B 0,C 180,E1 -27872.53,E2 -27872.53} C_VEL
LIN {X 0,Y 110.505,Z 516.411,A -85,B 0,C 180,E1 -27876.224,E2 -27876.224} C_VEL
LIN {X 0,Y 110.15,Z 510.364,A -85,B 0,C 180,E1 -27881.396,E2 -27881.396} C_VEL
LIN {X 0,Y 110.115,Z 508.329,A -85,B 0,C 180,E1 -27883.211,E2 -27883.211} C_VEL
LIN {X 0,Y 109.527,Z 501.91,A -85,B 0,C 180,E1 -27890.769,E2 -27890.769} C_VEL
LIN {X 0,Y 109.335,Z 500.842,A -85,B 0,C 180,E1 -27892.614,E2 -27892.614} C_VEL
LIN {X 0,Y 108.835,Z 498.089,A -85,B 0,C 180,E1 -27900,E2 -27900} C_VEL
LIN {X 0,Y 108.001,Z 499.046,A -85,B 0,C 180,E1 -27907.478,E2 -27907.478} C_VEL
LIN {X 0,Y 108.13,Z 500.304,A -85,B 0,C 180,E1 -27912.853,E2 -27912.853} C_VEL
LIN {X 0,Y 108.509,Z 502.818,A -85,B 0,C 180,E1 -27918.896,E2 -27918.896} C_VEL
LIN {X 0,Y 109.038,Z 506.905,A -85,B 0,C 180,E1 -27925.528,E2 -27925.528} C_VEL
LIN {X 0,Y 109.35,Z 511.075,A -85,B 0,C 180,E1 -27930.942,E2 -27930.942} C_VEL
LIN {X 0,Y 109.527,Z 514.765,A -85,B 0,C 180,E1 -27935.275,E2 -27935.275} C_VEL
LIN {X 0,Y 109.26,Z 519.297,A -85,B 0,C 180,E1 -27940.034,E2 -27940.034} C_VEL
LIN {X 0,Y 108.788,Z 522.83,A -85,B 0,C 180,E1 -27943.636,E2 -27943.636} C_VEL
LIN {X 0,Y 108.201,Z 523.856,A -85,B 0,C 180,E1 -27944.398,E2 -27944.398} C_VEL
LIN {X 0,Y 101.807,Z 531.134,A -85,B 0,C 180,E1 -27949.018,E2 -27949.018} C_VEL
LIN {X 0,Y 96.184,Z 536.94,A -85,B 0,C 180,E1 -27954.228,E2 -27954.228} C_VEL
LIN {X 0,Y 91.225,Z 541.533,A -85,B 0,C 180,E1 -27959.949,E2 -27959.949} C_VEL
LIN {X 0,Y 88.532,Z 543.849,A -85,B 0,C 180,E1 -27963.767,E2 -27963.767} C_VEL
LIN {X 0,Y 85.961,Z 545.651,A -85,B 0,C 180,E1 -27967.044,E2 -27967.044} C_VEL
LIN {X 0,Y 80.47,Z 548.163,A -85,B 0,C 180,E1 -27972.457,E2 -27972.457} C_VEL
LIN {X 0,Y 75.661,Z 550.027,A -85,B 0,C 180,E1 -27978.698,E2 -27978.698} C_VEL
LIN {X 0,Y 74.311,Z 550.603,A -85,B 0,C 180,E1 -27983.063,E2 -27983.063} C_VEL
LIN {X 0,Y 73.937,Z 550.976,A -85,B 0,C 180,E1 -27990,E2 -27990} C_VEL
LIN {X 0,Y 74.189,Z 550.786,A -85,B 0,C 180,E1 -27995.435,E2 -27995.435} C_VEL
LIN {X 0,Y 76.162,Z 549.303,A -85,B 0,C 180,E1 -28006.071,E2 -28006.071} C_VEL
LIN {X 0,Y 78.14,Z 547.966,A -85,B 0,C 180,E1 -28011.085,E2 -28011.085} C_VEL
LIN {X 0,Y 82.08,Z 545.136,A -85,B 0,C 180,E1 -28018.094,E2 -28018.094} C_VEL
LIN {X 0,Y 86.929,Z 541.309,A -85,B 0,C 180,E1 -28024.467,E2 -28024.467} C_VEL
LIN {X 0,Y 93.475,Z 535.373,A -85,B 0,C 180,E1 -28031.248,E2 -28031.248} C_VEL
LIN {X 0,Y 99.903,Z 528.973,A -85,B 0,C 180,E1 -28036.143,E2 -28036.143} C_VEL
LIN {X 0,Y 102.177,Z 526.493,A -85,B 0,C 180,E1 -28037.682,E2 -28037.682} C_VEL
LIN {X 0,Y 103.106,Z 525.221,A -85,B 0,C 180,E1 -28038.572,E2 -28038.572} C_VEL
LIN {X 0,Y 103.971,Z 520.372,A -85,B 0,C 180,E1 -28044.208,E2 -28044.208} C_VEL
LIN {X 0,Y 104.244,Z 516.12,A -85,B 0,C 180,E1 -28049.628,E2 -28049.628} C_VEL
LIN {X 0,Y 104.35,Z 511.622,A -85,B 0,C 180,E1 -28056.165,E2 -28056.165} C_VEL
LIN {X 0,Y 104.275,Z 509.133,A -85,B 0,C 180,E1 -28060.662,E2 -28060.662} C_VEL
LIN {X 0,Y 104.182,Z 507.528,A -85,B 0,C 180,E1 -28064.345,E2 -28064.345} C_VEL
LIN {X 0,Y 104.251,Z 506.148,A -85,B 0,C 180,E1 -28068.332,E2 -28068.332} C_VEL
LIN {X 0,Y 104.64,Z 504.783,A -85,B 0,C 180,E1 -28076.149,E2 -28076.149} C_VEL
LIN {X 0,Y 105.219,Z 504.584,A -85,B 0,C 180,E1 -28080,E2 -28080} C_VEL
LIN {X 0,Y 105.358,Z 505.726,A -85,B 0,C 180,E1 -28083.825,E2 -28083.825} C_VEL
LIN {X 0,Y 105.624,Z 507.373,A -85,B 0,C 180,E1 -28087.647,E2 -28087.647} C_VEL
LIN {X 0,Y 105.663,Z 513.485,A -85,B 0,C 180,E1 -28095.429,E2 -28095.429} C_VEL
LIN {X 0,Y 105.582,Z 518.756,A -85,B 0,C 180,E1 -28100.555,E2 -28100.555} C_VEL
LIN {X 0,Y 105.169,Z 524.938,A -85,B 0,C 180,E1 -28105.714,E2 -28105.714} C_VEL
LIN {X 0,Y 104.717,Z 527.155,A -85,B 0,C 180,E1 -28107.289,E2 -28107.289} C_VEL
LIN {X 0,Y 100.629,Z 534.852,A -85,B 0,C 180,E1 -28111.18,E2 -28111.18} C_VEL
LIN {X 0,Y 94.873,Z 543.892,A -85,B 0,C 180,E1 -28116.581,E2 -28116.581} C_VEL
LIN {X 0,Y 89.653,Z 550.894,A -85,B 0,C 180,E1 -28121.866,E2 -28121.866} C_VEL
LIN {X 0,Y 84.272,Z 557.251,A -85,B 0,C 180,E1 -28128.151,E2 -28128.151} C_VEL
LIN {X 0,Y 79.014,Z 562.181,A -85,B 0,C 180,E1 -28134.68,E2 -28134.68} C_VEL
LIN {X 0,Y 74.94,Z 566.005,A -85,B 0,C 180,E1 -28142.037,E2 -28142.037} C_VEL
LIN {X 0,Y 73.112,Z 568.034,A -85,B 0,C 180,E1 -28147.387,E2 -28147.387} C_VEL
LIN {X 0,Y 71.51,Z 570.773,A -85,B 0,C 180,E1 -28158.665,E2 -28158.665} C_VEL
LIN {X 0,Y 71.743,Z 571.556,A -85,B 0,C 180,E1 -28164.379,E2 -28164.379} C_VEL
LIN {X 0,Y 72.456,Z 571.913,A -85,B 0,C 180,E1 -28170,E2 -28170} C_VEL
LIN {X 0,Y 71.503,Z 570.869,A -85,B 0,C 180,E1 -28180.613,E2 -28180.613} C_VEL
LIN {X 0,Y 71.949,Z 569.56,A -85,B 0,C 180,E1 -28187.041,E2 -28187.041} C_VEL
LIN {X 0,Y 73.94,Z 566.992,A -85,B 0,C 180,E1 -28195.324,E2 -28195.324} C_VEL
LIN {X 0,Y 77.505,Z 563.465,A -85,B 0,C 180,E1 -28202.962,E2 -28202.962} C_VEL
LIN {X 0,Y 82.81,Z 558.538,A -85,B 0,C 180,E1 -28210.198,E2 -28210.198} C_VEL
LIN {X 0,Y 87.815,Z 553.018,A -85,B 0,C 180,E1 -28216.079,E2 -28216.079} C_VEL
LIN {X 0,Y 93.495,Z 545.62,A -85,B 0,C 180,E1 -28222.119,E2 -28222.119} C_VEL
LIN {X 0,Y 98.544,Z 538.053,A -85,B 0,C 180,E1 -28226.929,E2 -28226.929} C_VEL
LIN {X 0,Y 103.686,Z 528.864,A -85,B 0,C 180,E1 -28231.784,E2 -28231.784} C_VEL
LIN {X 0,Y 104.777,Z 526.603,A -85,B 0,C 180,E1 -28232.863,E2 -28232.863} C_VEL
LIN {X 0,Y 105.397,Z 520.476,A -85,B 0,C 180,E1 -28237.688,E2 -28237.688} C_VEL
LIN {X 0,Y 105.517,Z 514.041,A -85,B 0,C 180,E1 -28243.728,E2 -28243.728} C_VEL
LIN {X 0,Y 105.404,Z 511.642,A -85,B 0,C 180,E1 -28246.505,E2 -28246.505} C_VEL
LIN {X 0,Y 105.468,Z 507.141,A -85,B 0,C 180,E1 -28252.341,E2 -28252.341} C_VEL
LIN {X 0,Y 105.21,Z 505.47,A -85,B 0,C 180,E1 -28256.17,E2 -28256.17} C_VEL
LIN {X 0,Y 105.13,Z 504.222,A -85,B 0,C 180,E1 -28260,E2 -28260} C_VEL
LIN {X 0,Y 104.136,Z 505.079,A -85,B 0,C 180,E1 -28267.758,E2 -28267.758} C_VEL
LIN {X 0,Y 104.106,Z 505.875,A -85,B 0,C 180,E1 -28271.685,E2 -28271.685} C_VEL
LIN {X 0,Y 104.071,Z 507.214,A -85,B 0,C 180,E1 -28275.672,E2 -28275.672} C_VEL
LIN {X 0,Y 104.17,Z 509.012,A -85,B 0,C 180,E1 -28279.715,E2 -28279.715} C_VEL
LIN {X 0,Y 104.216,Z 512.354,A -85,B 0,C 180,E1 -28285.428,E2 -28285.428} C_VEL
LIN {X 0,Y 104.154,Z 515.854,A -85,B 0,C 180,E1 -28290.401,E2 -28290.401} C_VEL
LIN {X 0,Y 103.881,Z 520.048,A -85,B 0,C 180,E1 -28295.722,E2 -28295.722} C_VEL
LIN {X 0,Y 103.03,Z 524.945,A -85,B 0,C 180,E1 -28301.379,E2 -28301.379} C_VEL
LIN {X 0,Y 102.223,Z 526.191,A -85,B 0,C 180,E1 -28302.346,E2 -28302.346} C_VEL
LIN {X 0,Y 95.544,Z 533.229,A -85,B 0,C 180,E1 -28307.124,E2 -28307.124} C_VEL
LIN {X 0,Y 90.577,Z 537.947,A -85,B 0,C 180,E1 -28311.63,E2 -28311.63} C_VEL
LIN {X 0,Y 85.215,Z 542.539,A -85,B 0,C 180,E1 -28317.582,E2 -28317.582} C_VEL
LIN {X 0,Y 80.645,Z 546.061,A -85,B 0,C 180,E1 -28324.167,E2 -28324.167} C_VEL
LIN {X 0,Y 78.16,Z 547.879,A -85,B 0,C 180,E1 -28328.919,E2 -28328.919} C_VEL
LIN {X 0,Y 76.175,Z 549.244,A -85,B 0,C 180,E1 -28333.931,E2 -28333.931} C_VEL
LIN {X 0,Y 74.311,Z 550.603,A -85,B 0,C 180,E1 -28343.063,E2 -28343.063} C_VEL
LIN {X 0,Y 73.756,Z 550.914,A -85,B 0,C 180,E1 -28346.075,E2 -28346.075} C_VEL
LIN {X 0,Y 72.275,Z 551.281,A -85,B 0,C 180,E1 -28350.58,E2 -28350.58} C_VEL
LIN {X 0,Y 69.61,Z 551.418,A -85,B 0,C 180,E1 -28358.354,E2 -28358.354} C_VEL
LIN {X 0,Y 68.929,Z 550.826,A -85,B 0,C 180,E1 -28364.899,E2 -28364.899} C_VEL
LIN {X 0,Y 69.576,Z 550.209,A -85,B 0,C 180,E1 -28368.09,E2 -28368.09} C_VEL
LIN {X 0,Y 71.627,Z 548.971,A -85,B 0,C 180,E1 -28373.108,E2 -28373.108} C_VEL
LIN {X 0,Y 75.953,Z 546.14,A -85,B 0,C 180,E1 -28380.592,E2 -28380.592} C_VEL
LIN {X 0,Y 81.232,Z 542.313,A -85,B 0,C 180,E1 -28387.273,E2 -28387.273} C_VEL
LIN {X 0,Y 88.322,Z 536.369,A -85,B 0,C 180,E1 -28394.261,E2 -28394.261} C_VEL
LIN {X 0,Y 96.376,Z 528.774,A -85,B 0,C 180,E1 -28399.968,E2 -28399.968} C_VEL
LIN {X 0,Y 97.398,Z 527.538,A -85,B 0,C 180,E1 -28400.868,E2 -28400.868} C_VEL
LIN {X 0,Y 98.242,Z 524.302,A -85,B 0,C 180,E1 -28405.089,E2 -28405.089} C_VEL
LIN {X 0,Y 98.819,Z 520.763,A -85,B 0,C 180,E1 -28410.143,E2 -28410.143} C_VEL
LIN {X 0,Y 99.391,Z 516.604,A -85,B 0,C 180,E1 -28416.814,E2 -28416.814} C_VEL
LIN {X 0,Y 99.533,Z 515.232,A -85,B 0,C 180,E1 -28419.326,E2 -28419.326} C_VEL
LIN {X 0,Y 99.636,Z 513.46,A -85,B 0,C 180,E1 -28423.611,E2 -28423.611} C_VEL
LIN {X 0,Y 99.953,Z 511.546,A -85,B 0,C 180,E1 -28429.861,E2 -28429.861} C_VEL
LIN {X 0,Y 100.488,Z 510.632,A -85,B 0,C 180,E1 -28435.989,E2 -28435.989} C_VEL
LIN {X 0,Y 101.129,Z 510.45,A -85,B 0,C 180,E1 -28440,E2 -28440} C_VEL
LIN {X 0,Y 101.199,Z 511.683,A -85,B 0,C 180,E1 -28443.982,E2 -28443.982} C_VEL
LIN {X 0,Y 101.22,Z 513.64,A -85,B 0,C 180,E1 -28447.982,E2 -28447.982} C_VEL
LIN {X 0,Y 100.917,Z 518.19,A -85,B 0,C 180,E1 -28454.105,E2 -28454.105} C_VEL
LIN {X 0,Y 100.421,Z 523.241,A -85,B 0,C 180,E1 -28459.416,E2 -28459.416} C_VEL
LIN {X 0,Y 99.691,Z 528.317,A -85,B 0,C 180,E1 -28464.049,E2 -28464.049} C_VEL
LIN {X 0,Y 99.074,Z 529.941,A -85,B 0,C 180,E1 -28465.19,E2 -28465.19} C_VEL
LIN {X 0,Y 94.577,Z 537.199,A -85,B 0,C 180,E1 -28469.174,E2 -28469.174} C_VEL
LIN {X 0,Y 87.842,Z 546.283,A -85,B 0,C 180,E1 -28475.226,E2 -28475.226} C_VEL
LIN {X 0,Y 81.845,Z 553.198,A -85,B 0,C 180,E1 -28481.292,E2 -28481.292} C_VEL
LIN {X 0,Y 77.041,Z 558.017,A -85,B 0,C 180,E1 -28486.869,E2 -28486.869} C_VEL
LIN {X 0,Y 71.619,Z 562.541,A -85,B 0,C 180,E1 -28493.93,E2 -28493.93} C_VEL
LIN {X 0,Y 67.523,Z 566.032,A -85,B 0,C 180,E1 -28502.072,E2 -28502.072} C_VEL
LIN {X 0,Y 65.145,Z 568.577,A -85,B 0,C 180,E1 -28511.117,E2 -28511.117} C_VEL
LIN {X 0,Y 64.631,Z 570.533,A -85,B 0,C 180,E1 -28523.758,E2 -28523.758} C_VEL
LIN {X 0,Y 65.341,Z 570.896,A -85,B 0,C 180,E1 -28530.001,E2 -28530.001} C_VEL
LIN {X 0,Y 64.451,Z 569.954,A -85,B 0,C 180,E1 -28541.068,E2 -28541.068} C_VEL
LIN {X 0,Y 65.139,Z 568.536,A -85,B 0,C 180,E1 -28548.886,E2 -28548.886} C_VEL
LIN {X 0,Y 67.513,Z 565.964,A -85,B 0,C 180,E1 -28557.934,E2 -28557.934} C_VEL
LIN {X 0,Y 71.602,Z 562.44,A -85,B 0,C 180,E1 -28566.081,E2 -28566.081} C_VEL
LIN {X 0,Y 76.886,Z 557.992,A -85,B 0,C 180,E1 -28573.008,E2 -28573.008} C_VEL
LIN {X 0,Y 81.868,Z 553.041,A -85,B 0,C 180,E1 -28578.691,E2 -28578.691} C_VEL
LIN {X 0,Y 86.96,Z 547.195,A -85,B 0,C 180,E1 -28583.92,E2 -28583.92} C_VEL
LIN {X 0,Y 93.433,Z 538.55,A -85,B 0,C 180,E1 -28589.887,E2 -28589.887} C_VEL
LIN {X 0,Y 98.969,Z 529.762,A -85,B 0,C 180,E1 -28594.781,E2 -28594.781} C_VEL
LIN {X 0,Y 99.671,Z 527.546,A -85,B 0,C 180,E1 -28596.444,E2 -28596.444} C_VEL
LIN {X 0,Y 100.299,Z 523.05,A -85,B 0,C 180,E1 -28600.559,E2 -28600.559} C_VEL
LIN {X 0,Y 100.826,Z 517.774,A -85,B 0,C 180,E1 -28606.085,E2 -28606.085} C_VEL
LIN {X 0,Y 101.117,Z 513.356,A -85,B 0,C 180,E1 -28612.01,E2 -28612.01} C_VEL
LIN {X 0,Y 101.059,Z 511.441,A -85,B 0,C 180,E1 -28616.012,E2 -28616.012} C_VEL
LIN {X 0,Y 101.046,Z 510.123,A -85,B 0,C 180,E1 -28620,E2 -28620} C_VEL
LIN {X 0,Y 99.941,Z 510.907,A -85,B 0,C 180,E1 -28628.085,E2 -28628.085} C_VEL
LIN {X 0,Y 99.709,Z 511.772,A -85,B 0,C 180,E1 -28632.208,E2 -28632.208} C_VEL
LIN {X 0,Y 99.531,Z 513.167,A -85,B 0,C 180,E1 -28636.406,E2 -28636.406} C_VEL
LIN {X 0,Y 99.369,Z 515.034,A -85,B 0,C 180,E1 -28640.71,E2 -28640.71} C_VEL
LIN {X 0,Y 99.135,Z 517.482,A -85,B 0,C 180,E1 -28645.174,E2 -28645.174} C_VEL
LIN {X 0,Y 98.549,Z 522.174,A -85,B 0,C 180,E1 -28652.332,E2 -28652.332} C_VEL
LIN {X 0,Y 97.629,Z 526.161,A -85,B 0,C 180,E1 -28657.64,E2 -28657.64} C_VEL
LIN {X 0,Y 97.318,Z 527.268,A -85,B 0,C 180,E1 -28659.073,E2 -28659.073} C_VEL
LIN {X 0,Y 96.389,Z 528.507,A -85,B 0,C 180,E1 -28660.04,E2 -28660.04} C_VEL
LIN {X 0,Y 88.845,Z 535.726,A -85,B 0,C 180,E1 -28665.393,E2 -28665.393} C_VEL
LIN {X 0,Y 83.195,Z 540.601,A -85,B 0,C 180,E1 -28670.685,E2 -28670.685} C_VEL
LIN {X 0,Y 77.564,Z 544.836,A -85,B 0,C 180,E1 -28677.067,E2 -28677.067} C_VEL
LIN {X 0,Y 74.383,Z 547.067,A -85,B 0,C 180,E1 -28681.808,E2 -28681.808} C_VEL
LIN {X 0,Y 71.647,Z 548.885,A -85,B 0,C 180,E1 -28686.898,E2 -28686.898} C_VEL
LIN {X 0,Y 69.449,Z 550.249,A -85,B 0,C 180,E1 -28692.326,E2 -28692.326} C_VEL
LIN {X 0,Y 67.197,Z 551.765,A -85,B 0,C 180,E1 -28703.996,E2 -28703.996} C_VEL
LIN {X 0,Y 66.909,Z 551.981,A -85,B 0,C 180,E1 -28709.999,E2 -28709.999} C_VEL
LIN {X 0,Y 67.196,Z 551.791,A -85,B 0,C 180,E1 -28716.003,E2 -28716.003} C_VEL
LIN {X 0,Y 69.436,Z 550.308,A -85,B 0,C 180,E1 -28727.676,E2 -28727.676} C_VEL
LIN {X 0,Y 69.576,Z 550.209,A -85,B 0,C 180,E1 -28728.09,E2 -28728.09} C_VEL
LIN {X 0,Y 70.752,Z 549.221,A -85,B 0,C 180,E1 -28732.737,E2 -28732.737} C_VEL
LIN {X 0,Y 71.956,Z 547.27,A -85,B 0,C 180,E1 -28740.495,E2 -28740.495} C_VEL
LIN {X 0,Y 73.545,Z 545.289,A -85,B 0,C 180,E1 -28746.436,E2 -28746.436} C_VEL
LIN {X 0,Y 75.749,Z 543.351,A -85,B 0,C 180,E1 -28750.386,E2 -28750.386} C_VEL
LIN {X 0,Y 76.739,Z 542.582,A -85,B 0,C 180,E1 -28751.538,E2 -28751.538} C_VEL
LIN {X 0,Y 84.524,Z 536.472,A -85,B 0,C 180,E1 -28758.446,E2 -28758.446} C_VEL
LIN {X 0,Y 90.747,Z 530.976,A -85,B 0,C 180,E1 -28762.544,E2 -28762.544} C_VEL
LIN {X 0,Y 91.798,Z 529.829,A -85,B 0,C 180,E1 -28763.501,E2 -28763.501} C_VEL
LIN {X 0,Y 92.779,Z 526.891,A -85,B 0,C 180,E1 -28767.977,E2 -28767.977} C_VEL
LIN {X 0,Y 93.757,Z 523.203,A -85,B 0,C 180,E1 -28774.095,E2 -28774.095} C_VEL
LIN {X 0,Y 94.314,Z 521.069,A -85,B 0,C 180,E1 -28778.124,E2 -28778.124} C_VEL
LIN {X 0,Y 94.874,Z 518.538,A -85,B 0,C 180,E1 -28784.365,E2 -28784.365} C_VEL
LIN {X 0,Y 95.504,Z 516.751,A -85,B 0,C 180,E1 -28791.536,E2 -28791.536} C_VEL
LIN {X 0,Y 96.028,Z 516.242,A -85,B 0,C 180,E1 -28795.803,E2 -28795.803} C_VEL
LIN {X 0,Y 96.705,Z 516.107,A -85,B 0,C 180,E1 -28800,E2 -28800} C_VEL
LIN {X 0,Y 96.663,Z 517.472,A -85,B 0,C 180,E1 -28804.169,E2 -28804.169} C_VEL
LIN {X 0,Y 96.602,Z 518.438,A -85,B 0,C 180,E1 -28806.265,E2 -28806.265} C_VEL
LIN {X 0,Y 95.989,Z 522.67,A -85,B 0,C 180,E1 -28812.688,E2 -28812.688} C_VEL
LIN {X 0,Y 95.055,Z 527.591,A -85,B 0,C 180,E1 -28818.314,E2 -28818.314} C_VEL
LIN {X 0,Y 94.241,Z 531.169,A -85,B 0,C 180,E1 -28821.893,E2 -28821.893} C_VEL
LIN {X 0,Y 92.228,Z 534.372,A -85,B 0,C 180,E1 -28823.876,E2 -28823.876} C_VEL
LIN {X 0,Y 85.944,Z 542.596,A -85,B 0,C 180,E1 -28829.059,E2 -28829.059} C_VEL
LIN {X 0,Y 79.386,Z 549.967,A -85,B 0,C 180,E1 -28835.026,E2 -28835.026} C_VEL
LIN {X 0,Y 74.012,Z 555.16,A -85,B 0,C 180,E1 -28840.566,E2 -28840.566} C_VEL
LIN {X 0,Y 69.893,Z 558.64,A -85,B 0,C 180,E1 -28845.262,E2 -28845.262} C_VEL
LIN {X 0,Y 64.245,Z 562.816,A -85,B 0,C 180,E1 -28853.011,E2 -28853.011} C_VEL
LIN {X 0,Y 60.109,Z 565.981,A -85,B 0,C 180,E1 -28862.116,E2 -28862.116} C_VEL
LIN {X 0,Y 57.537,Z 568.726,A -85,B 0,C 180,E1 -28875.86,E2 -28875.86} C_VEL
LIN {X 0,Y 57.528,Z 569.511,A -85,B 0,C 180,E1 -28882.983,E2 -28882.983} C_VEL
LIN {X 0,Y 58.225,Z 569.878,A -85,B 0,C 180,E1 -28890.001,E2 -28890.001} C_VEL
LIN {X 0,Y 57.423,Z 569.028,A -85,B 0,C 180,E1 -28901.731,E2 -28901.731} C_VEL
LIN {X 0,Y 58.397,Z 567.509,A -85,B 0,C 180,E1 -28911.165,E2 -28911.165} C_VEL
LIN {X 0,Y 61.271,Z 564.938,A -85,B 0,C 180,E1 -28921.076,E2 -28921.076} C_VEL
LIN {X 0,Y 65.944,Z 561.413,A -85,B 0,C 180,E1 -28929.752,E2 -28929.752} C_VEL
LIN {X 0,Y 72.204,Z 556.608,A -85,B 0,C 180,E1 -28937.414,E2 -28937.414} C_VEL
LIN {X 0,Y 78.255,Z 550.892,A -85,B 0,C 180,E1 -28943.929,E2 -28943.929} C_VEL
LIN {X 0,Y 83.973,Z 544.677,A -85,B 0,C 180,E1 -28949.265,E2 -28949.265} C_VEL
LIN {X 0,Y 89.782,Z 537.434,A -85,B 0,C 180,E1 -28954.187,E2 -28954.187} C_VEL
LIN {X 0,Y 93.062,Z 532.832,A -85,B 0,C 180,E1 -28956.872,E2 -28956.872} C_VEL
LIN {X 0,Y 94.122,Z 531.003,A -85,B 0,C 180,E1 -28958.078,E2 -28958.078} C_VEL
LIN {X 0,Y 95.162,Z 526.345,A -85,B 0,C 180,E1 -28962.818,E2 -28962.818} C_VEL
LIN {X 0,Y 95.874,Z 522.457,A -85,B 0,C 180,E1 -28967.296,E2 -28967.296} C_VEL
LIN {X 0,Y 96.497,Z 518.177,A -85,B 0,C 180,E1 -28973.728,E2 -28973.728} C_VEL
LIN {X 0,Y 96.635,Z 515.794,A -85,B 0,C 180,E1 -28980,E2 -28980} C_VEL
LIN {X 0,Y 95.524,Z 516.306,A -85,B 0,C 180,E1 -28986.932,E2 -28986.932} C_VEL
LIN {X 0,Y 94.966,Z 517.44,A -85,B 0,C 180,E1 -28992.828,E2 -28992.828} C_VEL
LIN {X 0,Y 94.565,Z 518.919,A -85,B 0,C 180,E1 -28997.294,E2 -28997.294} C_VEL
LIN {X 0,Y 94.2,Z 520.839,A -85,B 0,C 180,E1 -29001.903,E2 -29001.903} C_VEL
LIN {X 0,Y 93.548,Z 523.469,A -85,B 0,C 180,E1 -29006.793,E2 -29006.793} C_VEL
LIN {X 0,Y 92.723,Z 526.653,A -85,B 0,C 180,E1 -29012.044,E2 -29012.044} C_VEL
LIN {X 0,Y 91.733,Z 529.585,A -85,B 0,C 180,E1 -29016.442,E2 -29016.442} C_VEL
LIN {X 0,Y 90.749,Z 530.717,A -85,B 0,C 180,E1 -29017.456,E2 -29017.456} C_VEL
LIN {X 0,Y 83.958,Z 536.755,A -85,B 0,C 180,E1 -29022.042,E2 -29022.042} C_VEL
LIN {X 0,Y 77.886,Z 541.607,A -85,B 0,C 180,E1 -29027.409,E2 -29027.409} C_VEL
LIN {X 0,Y 71.768,Z 545.842,A -85,B 0,C 180,E1 -29034.015,E2 -29034.015} C_VEL
LIN {X 0,Y 68.27,Z 548.073,A -85,B 0,C 180,E1 -29039.02,E2 -29039.02} C_VEL
LIN {X 0,Y 65.241,Z 549.891,A -85,B 0,C 180,E1 -29044.475,E2 -29044.475} C_VEL
LIN {X 0,Y 62.789,Z 551.255,A -85,B 0,C 180,E1 -29050.379,E2 -29050.379} C_VEL
LIN {X 0,Y 60.212,Z 552.77,A -85,B 0,C 180,E1 -29063.297,E2 -29063.297} C_VEL
LIN {X 0,Y 59.881,Z 552.986,A -85,B 0,C 180,E1 -29069.999,E2 -29069.999} C_VEL
LIN {X 0,Y 60.211,Z 552.795,A -85,B 0,C 180,E1 -29076.703,E2 -29076.703} C_VEL
LIN {X 0,Y 62.776,Z 551.313,A -85,B 0,C 180,E1 -29089.624,E2 -29089.624} C_VEL
LIN {X 0,Y 65.222,Z 549.976,A -85,B 0,C 180,E1 -29095.532,E2 -29095.532} C_VEL
LIN {X 0,Y 69.994,Z 547.144,A -85,B 0,C 180,E1 -29103.521,E2 -29103.521} C_VEL
LIN {X 0,Y 76.739,Z 542.582,A -85,B 0,C 180,E1 -29111.538,E2 -29111.538} C_VEL
LIN {X 0,Y 79.669,Z 540.207,A -85,B 0,C 180,E1 -29114.939,E2 -29114.939} C_VEL
LIN {X 0,Y 82.802,Z 536.95,A -85,B 0,C 180,E1 -29119.598,E2 -29119.598} C_VEL
LIN {X 0,Y 84.663,Z 534.501,A -85,B 0,C 180,E1 -29123.154,E2 -29123.154} C_VEL
LIN {X 0,Y 86.556,Z 531.362,A -85,B 0,C 180,E1 -29127.966,E2 -29127.966} C_VEL
LIN {X 0,Y 87.249,Z 529.9,A -85,B 0,C 180,E1 -29130.415,E2 -29130.415} C_VEL
LIN {X 0,Y 88.11,Z 527.918,A -85,B 0,C 180,E1 -29134.144,E2 -29134.144} C_VEL
LIN {X 0,Y 89.221,Z 524.893,A -85,B 0,C 180,E1 -29140.953,E2 -29140.953} C_VEL
LIN {X 0,Y 90.008,Z 523.092,A -85,B 0,C 180,E1 -29146.453,E2 -29146.453} C_VEL
LIN {X 0,Y 90.554,Z 522.121,A -85,B 0,C 180,E1 -29151.07,E2 -29151.07} C_VEL
LIN {X 0,Y 91.483,Z 521.519,A -85,B 0,C 180,E1 -29157.078,E2 -29157.078} C_VEL
LIN {X 0,Y 91.973,Z 521.52,A -85,B 0,C 180,E1 -29160,E2 -29160} C_VEL
LIN {X 0,Y 91.752,Z 523.386,A -85,B 0,C 180,E1 -29165.271,E2 -29165.271} C_VEL
LIN {X 0,Y 90.88,Z 526.926,A -85,B 0,C 180,E1 -29171.147,E2 -29171.147} C_VEL
LIN {X 0,Y 89.723,Z 530.997,A -85,B 0,C 180,E1 -29176.31,E2 -29176.31} C_VEL
LIN {X 0,Y 89.052,Z 533.126,A -85,B 0,C 180,E1 -29178.73,E2 -29178.73} C_VEL
LIN {X 0,Y 88.281,Z 534.614,A -85,B 0,C 180,E1 -29180.01,E2 -29180.01} C_VEL
LIN {X 0,Y 82.124,Z 541.923,A -85,B 0,C 180,E1 -29184.687,E2 -29184.687} C_VEL
LIN {X 0,Y 75.354,Z 548.902,A -85,B 0,C 180,E1 -29190.377,E2 -29190.377} C_VEL
LIN {X 0,Y 69.451,Z 554.109,A -85,B 0,C 180,E1 -29195.949,E2 -29195.949} C_VEL
LIN {X 0,Y 64.972,Z 557.61,A -85,B 0,C 180,E1 -29200.784,E2 -29200.784} C_VEL
LIN {X 0,Y 58.674,Z 561.791,A -85,B 0,C 180,E1 -29208.792,E2 -29208.792} C_VEL
LIN {X 0,Y 53.884,Z 564.958,A -85,B 0,C 180,E1 -29218.553,E2 -29218.553} C_VEL
LIN {X 0,Y 50.626,Z 567.702,A -85,B 0,C 180,E1 -29233.881,E2 -29233.881} C_VEL
LIN {X 0,Y 50.442,Z 568.489,A -85,B 0,C 180,E1 -29241.992,E2 -29241.992} C_VEL
LIN {X 0,Y 51.108,Z 568.86,A -85,B 0,C 180,E1 -29250.001,E2 -29250.001} C_VEL
LIN {X 0,Y 50.397,Z 568.094,A -85,B 0,C 180,E1 -29262.532,E2 -29262.532} C_VEL
LIN {X 0,Y 51.764,Z 566.481,A -85,B 0,C 180,E1 -29274.037,E2 -29274.037} C_VEL
LIN {X 0,Y 55.245,Z 563.91,A -85,B 0,C 180,E1 -29284.923,E2 -29284.923} C_VEL
LIN {X 0,Y 60.612,Z 560.388,A -85,B 0,C 180,E1 -29294.085,E2 -29294.085} C_VEL
LIN {X 0,Y 66.972,Z 555.959,A -85,B 0,C 180,E1 -29301.427,E2 -29301.427} C_VEL
LIN {X 0,Y 74.115,Z 549.826,A -85,B 0,C 180,E1 -29308.588,E2 -29308.588} C_VEL
LIN {X 0,Y 80.657,Z 543.267,A -85,B 0,C 180,E1 -29314.172,E2 -29314.172} C_VEL
LIN {X 0,Y 86.664,Z 536.313,A -85,B 0,C 180,E1 -29318.844,E2 -29318.844} C_VEL
LIN {X 0,Y 88.174,Z 534.451,A -85,B 0,C 180,E1 -29319.965,E2 -29319.965} C_VEL
LIN {X 0,Y 89.261,Z 531.948,A -85,B 0,C 180,E1 -29322.362,E2 -29322.362} C_VEL
LIN {X 0,Y 90.266,Z 528.529,A -85,B 0,C 180,E1 -29326.492,E2 -29326.492} C_VEL
LIN {X 0,Y 90.775,Z 526.719,A -85,B 0,C 180,E1 -29328.84,E2 -29328.84} C_VEL
LIN {X 0,Y 91.699,Z 522.953,A -85,B 0,C 180,E1 -29335.11,E2 -29335.11} C_VEL
LIN {X 0,Y 91.908,Z 521.229,A -85,B 0,C 180,E1 -29340,E2 -29340} C_VEL
LIN {X 0,Y 90.727,Z 521.618,A -85,B 0,C 180,E1 -29346.659,E2 -29346.659} C_VEL
LIN {X 0,Y 89.931,Z 522.832,A -85,B 0,C 180,E1 -29353.559,E2 -29353.559} C_VEL
LIN {X 0,Y 89.136,Z 524.607,A -85,B 0,C 180,E1 -29358.887,E2 -29358.887} C_VEL
LIN {X 0,Y 88.498,Z 526.455,A -85,B 0,C 180,E1 -29363.395,E2 -29363.395} C_VEL
LIN {X 0,Y 87.388,Z 529.254,A -85,B 0,C 180,E1 -29368.852,E2 -29368.852} C_VEL
LIN {X 0,Y 86.657,Z 531.031,A -85,B 0,C 180,E1 -29372.006,E2 -29372.006} C_VEL
LIN {X 0,Y 85.296,Z 532.931,A -85,B 0,C 180,E1 -29374.516,E2 -29374.516} C_VEL
LIN {X 0,Y 77.764,Z 539.105,A -85,B 0,C 180,E1 -29379.611,E2 -29379.611} C_VEL
LIN {X 0,Y 70.608,Z 544.161,A -85,B 0,C 180,E1 -29385.832,E2 -29385.832} C_VEL
LIN {X 0,Y 64.268,Z 548.034,A -85,B 0,C 180,E1 -29393.025,E2 -29393.025} C_VEL
LIN {X 0,Y 58.977,Z 550.897,A -85,B 0,C 180,E1 -29401.532,E2 -29401.532} C_VEL
LIN {X 0,Y 56.218,Z 552.26,A -85,B 0,C 180,E1 -29407.973,E2 -29407.973} C_VEL
LIN {X 0,Y 53.239,Z 553.776,A -85,B 0,C 180,E1 -29422.414,E2 -29422.414} C_VEL
LIN {X 0,Y 52.853,Z 553.991,A -85,B 0,C 180,E1 -29429.999,E2 -29429.999} C_VEL
LIN {X 0,Y 53.237,Z 553.8,A -85,B 0,C 180,E1 -29437.585,E2 -29437.585} C_VEL
LIN {X 0,Y 56.206,Z 552.317,A -85,B 0,C 180,E1 -29452.031,E2 -29452.031} C_VEL
LIN {X 0,Y 58.958,Z 550.98,A -85,B 0,C 180,E1 -29458.477,E2 -29458.477} C_VEL
LIN {X 0,Y 64.252,Z 548.149,A -85,B 0,C 180,E1 -29466.984,E2 -29466.984} C_VEL
LIN {X 0,Y 71.482,Z 543.687,A -85,B 0,C 180,E1 -29475.123,E2 -29475.123} C_VEL
LIN {X 0,Y 78.863,Z 538.379,A -85,B 0,C 180,E1 -29481.404,E2 -29481.404} C_VEL
LIN {X 0,Y 85.288,Z 533.187,A -85,B 0,C 180,E1 -29485.49,E2 -29485.49} C_VEL
LIN {X 0,Y 86.729,Z 531.247,A -85,B 0,C 180,E1 -29487.963,E2 -29487.963} C_VEL
LIN {X 0,Y 87.249,Z 529.9,A -85,B 0,C 180,E1 -29490.415,E2 -29490.415} C_VEL
LIN {X 0,Y 87.564,Z 528.791,A -85,B 0,C 180,E1 -29492.875,E2 -29492.875} C_VEL
LIN {X 0,Y 87.288,Z 527.822,A -85,B 0,C 180,E1 -29496.701,E2 -29496.701} C_VEL
LIN {X 0,Y 86.546,Z 527.443,A -85,B 0,C 180,E1 -29500.602,E2 -29500.602} C_VEL
LIN {X 0,Y 85.441,Z 527.091,A -85,B 0,C 180,E1 -29511.569,E2 -29511.569} C_VEL
LIN {X 0,Y 86.099,Z 526.677,A -85,B 0,C 180,E1 -29515.318,E2 -29515.318} C_VEL
LIN {X 0,Y 86.915,Z 526.658,A -85,B 0,C 180,E1 -29520,E2 -29520} C_VEL
LIN {X 0,Y 86.535,Z 528.278,A -85,B 0,C 180,E1 -29524.658,E2 -29524.658} C_VEL
LIN {X 0,Y 85.564,Z 531.108,A -85,B 0,C 180,E1 -29529.721,E2 -29529.721} C_VEL
LIN {X 0,Y 84.207,Z 534.52,A -85,B 0,C 180,E1 -29534.5,E2 -29534.5} C_VEL
LIN {X 0,Y 83.649,Z 535.809,A -85,B 0,C 180,E1 -29536.117,E2 -29536.117} C_VEL
LIN {X 0,Y 82.613,Z 537.238,A -85,B 0,C 180,E1 -29537.283,E2 -29537.283} C_VEL
LIN {X 0,Y 74.499,Z 545.409,A -85,B 0,C 180,E1 -29543.106,E2 -29543.106} C_VEL
LIN {X 0,Y 67.935,Z 551.095,A -85,B 0,C 180,E1 -29548.437,E2 -29548.437} C_VEL
LIN {X 0,Y 60.52,Z 556.583,A -85,B 0,C 180,E1 -29555.621,E2 -29555.621} C_VEL
LIN {X 0,Y 53.494,Z 560.767,A -85,B 0,C 180,E1 -29563.732,E2 -29563.732} C_VEL
LIN {X 0,Y 47.906,Z 563.932,A -85,B 0,C 180,E1 -29574.069,E2 -29574.069} C_VEL
LIN {X 0,Y 43.796,Z 566.679,A -85,B 0,C 180,E1 -29591.281,E2 -29591.281} C_VEL
LIN {X 0,Y 43.353,Z 567.464,A -85,B 0,C 180,E1 -29600.671,E2 -29600.671} C_VEL
LIN {X 0,Y 43.989,Z 567.842,A -85,B 0,C 180,E1 -29610.001,E2 -29610.001} C_VEL
LIN {X 0,Y 43.401,Z 567.135,A -85,B 0,C 180,E1 -29623.693,E2 -29623.693} C_VEL
LIN {X 0,Y 45.319,Z 565.457,A -85,B 0,C 180,E1 -29637.727,E2 -29637.727} C_VEL
LIN {X 0,Y 49.542,Z 562.885,A -85,B 0,C 180,E1 -29649.671,E2 -29649.671} C_VEL
LIN {X 0,Y 55.693,Z 559.364,A -85,B 0,C 180,E1 -29659.215,E2 -29659.215} C_VEL
LIN {X 0,Y 60.747,Z 556.294,A -85,B 0,C 180,E1 -29664.658,E2 -29664.658} C_VEL
LIN {X 0,Y 67.921,Z 550.93,A -85,B 0,C 180,E1 -29671.586,E2 -29671.586} C_VEL
LIN {X 0,Y 75.826,Z 543.935,A -85,B 0,C 180,E1 -29677.952,E2 -29677.952} C_VEL
LIN {X 0,Y 82.539,Z 537.036,A -85,B 0,C 180,E1 -29682.729,E2 -29682.729} C_VEL
LIN {X 0,Y 83.585,Z 535.585,A -85,B 0,C 180,E1 -29683.907,E2 -29683.907} C_VEL
LIN {X 0,Y 84.93,Z 532.296,A -85,B 0,C 180,E1 -29688.303,E2 -29688.303} C_VEL
LIN {X 0,Y 85.519,Z 530.742,A -85,B 0,C 180,E1 -29690.54,E2 -29690.54} C_VEL
LIN {X 0,Y 86.448,Z 528.063,A -85,B 0,C 180,E1 -29695.337,E2 -29695.337} C_VEL
LIN {X 0,Y 86.862,Z 526.404,A -85,B 0,C 180,E1 -29700,E2 -29700} C_VEL
LIN {X 0,Y 85.689,Z 526.625,A -85,B 0,C 180,E1 -29706.285,E2 -29706.285} C_VEL
LIN {X 0,Y 85.216,Z 526.996,A -85,B 0,C 180,E1 -29709.494,E2 -29709.494} C_VEL
LIN {X 0,Y 84.379,Z 528.065,A -85,B 0,C 180,E1 -29714.47,E2 -29714.47} C_VEL
LIN {X 0,Y 83.093,Z 530.34,A -85,B 0,C 180,E1 -29721.505,E2 -29721.505} C_VEL
LIN {X 0,Y 82.248,Z 531.938,A -85,B 0,C 180,E1 -29725.293,E2 -29725.293} C_VEL
LIN {X 0,Y 80.997,Z 534.087,A -85,B 0,C 180,E1 -29729.808,E2 -29729.808} C_VEL
LIN {X 0,Y 80.117,Z 535.082,A -85,B 0,C 180,E1 -29731.208,E2 -29731.208} C_VEL
LIN {X 0,Y 73.459,Z 540.128,A -85,B 0,C 180,E1 -29735.398,E2 -29735.398} C_VEL
LIN {X 0,Y 65.75,Z 545.167,A -85,B 0,C 180,E1 -29741.562,E2 -29741.562} C_VEL
LIN {X 0,Y 58.806,Z 549.04,A -85,B 0,C 180,E1 -29748.904,E2 -29748.904} C_VEL
LIN {X 0,Y 52.905,Z 551.902,A -85,B 0,C 180,E1 -29757.901,E2 -29757.901} C_VEL
LIN {X 0,Y 49.773,Z 553.266,A -85,B 0,C 180,E1 -29764.937,E2 -29764.937} C_VEL
LIN {X 0,Y 46.282,Z 554.781,A -85,B 0,C 180,E1 -29781.265,E2 -29781.265} C_VEL
LIN {X 0,Y 45.825,Z 554.996,A -85,B 0,C 180,E1 -29789.999,E2 -29789.999} C_VEL
LIN {X 0,Y 46.28,Z 554.805,A -85,B 0,C 180,E1 -29798.734,E2 -29798.734} C_VEL
LIN {X 0,Y 49.76,Z 553.322,A -85,B 0,C 180,E1 -29815.068,E2 -29815.068} C_VEL
LIN {X 0,Y 52.886,Z 551.985,A -85,B 0,C 180,E1 -29822.11,E2 -29822.11} C_VEL
LIN {X 0,Y 58.791,Z 549.153,A -85,B 0,C 180,E1 -29831.108,E2 -29831.108} C_VEL
LIN {X 0,Y 65.707,Z 545.325,A -85,B 0,C 180,E1 -29838.479,E2 -29838.479} C_VEL
LIN {X 0,Y 74.676,Z 539.386,A -85,B 0,C 180,E1 -29845.619,E2 -29845.619} C_VEL
LIN {X 0,Y 80.109,Z 535.311,A -85,B 0,C 180,E1 -29848.8,E2 -29848.8} C_VEL
LIN {X 0,Y 81.047,Z 534.322,A -85,B 0,C 180,E1 -29850.129,E2 -29850.129} C_VEL
LIN {X 0,Y 82.332,Z 532.132,A -85,B 0,C 180,E1 -29854.735,E2 -29854.735} C_VEL
LIN {X 0,Y 83.504,Z 529.926,A -85,B 0,C 180,E1 -29860.326,E2 -29860.326} C_VEL
LIN {X 0,Y 84.455,Z 528.286,A -85,B 0,C 180,E1 -29865.543,E2 -29865.543} C_VEL
LIN {X 0,Y 85.441,Z 527.091,A -85,B 0,C 180,E1 -29871.569,E2 -29871.569} C_VEL
LIN {X 0,Y 85.297,Z 527.34,A -85,B 0,C 180,E1 -29874.182,E2 -29874.182} C_VEL
LIN {X 0,Y 84.492,Z 528.355,A -85,B 0,C 180,E1 -29876.714,E2 -29876.714} C_VEL
LIN {X 0,Y 80.726,Z 533.52,A -85,B 0,C 180,E1 -29885.228,E2 -29885.228} C_VEL
LIN {X 0,Y 80.231,Z 534.697,A -85,B 0,C 180,E1 -29887.55,E2 -29887.55} C_VEL
LIN {X 0,Y 78.926,Z 537.227,A -85,B 0,C 180,E1 -29891.623,E2 -29891.623} C_VEL
LIN {X 0,Y 77.763,Z 538.939,A -85,B 0,C 180,E1 -29893.698,E2 -29893.698} C_VEL
LIN {X 0,Y 68.967,Z 546.749,A -85,B 0,C 180,E1 -29899.505,E2 -29899.505} C_VEL
LIN {X 0,Y 61.947,Z 552,A -85,B 0,C 180,E1 -29904.823,E2 -29904.823} C_VEL
LIN {X 0,Y 56.088,Z 555.831,A -85,B 0,C 180,E1 -29910.08,E2 -29910.08} C_VEL
LIN {X 0,Y 46.479,Z 560.894,A -85,B 0,C 180,E1 -29920.885,E2 -29920.885} C_VEL
LIN {X 0,Y 42.298,Z 562.905,A -85,B 0,C 180,E1 -29928.348,E2 -29928.348} C_VEL
LIN {X 0,Y 37.067,Z 565.653,A -85,B 0,C 180,E1 -29947.716,E2 -29947.716} C_VEL
LIN {X 0,Y 36.303,Z 566.439,A -85,B 0,C 180,E1 -29958.838,E2 -29958.838} C_VEL
LIN {X 0,Y 36.868,Z 566.823,A -85,B 0,C 180,E1 -29970.001,E2 -29970.001} C_VEL
LIN {X 0,Y 37.05,Z 565.618,A -85,B 0,C 180,E1 -29992.297,E2 -29992.297} C_VEL
LIN {X 0,Y 42.289,Z 562.838,A -85,B 0,C 180,E1 -30011.665,E2 -30011.665} C_VEL
LIN {X 0,Y 48.81,Z 559.65,A -85,B 0,C 180,E1 -30022.368,E2 -30022.368} C_VEL
LIN {X 0,Y 56.582,Z 555.415,A -85,B 0,C 180,E1 -30030.398,E2 -30030.398} C_VEL
LIN {X 0,Y 64.711,Z 549.863,A -85,B 0,C 180,E1 -30037.394,E2 -30037.394} C_VEL
LIN {X 0,Y 73.305,Z 542.843,A -85,B 0,C 180,E1 -30043.484,E2 -30043.484} C_VEL
LIN {X 0,Y 77.743,Z 538.686,A -85,B 0,C 180,E1 -30046.364,E2 -30046.364} C_VEL
LIN {X 0,Y 79.324,Z 536.135,A -85,B 0,C 180,E1 -30049.794,E2 -30049.794} C_VEL
LIN {X 0,Y 80.732,Z 533.173,A -85,B 0,C 180,E1 -30055.006,E2 -30055.006} C_VEL
LIN {X 0,Y 81.475,Z 531.279,A -85,B 0,C 180,E1 -30060,E2 -30060} C_VEL
LIN {X 0,Y 80.434,Z 531.349,A -85,B 0,C 180,E1 -30065.679,E2 -30065.679} C_VEL
LIN {X 0,Y 79.164,Z 532.265,A -85,B 0,C 180,E1 -30072.427,E2 -30072.427} C_VEL
LIN {X 0,Y 78.433,Z 533.042,A -85,B 0,C 180,E1 -30075.594,E2 -30075.594} C_VEL
LIN {X 0,Y 77.137,Z 534.741,A -85,B 0,C 180,E1 -30081.373,E2 -30081.373} C_VEL
LIN {X 0,Y 76.622,Z 535.483,A -85,B 0,C 180,E1 -30083.474,E2 -30083.474} C_VEL
LIN {X 0,Y 75.252,Z 537.172,A -85,B 0,C 180,E1 -30087.47,E2 -30087.47} C_VEL
LIN {X 0,Y 66.695,Z 542.979,A -85,B 0,C 180,E1 -30092.54,E2 -30092.54} C_VEL
LIN {X 0,Y 58.66,Z 547.57,A -85,B 0,C 180,E1 -30098.851,E2 -30098.851} C_VEL
LIN {X 0,Y 51.354,Z 551.091,A -85,B 0,C 180,E1 -30106.821,E2 -30106.821} C_VEL
LIN {X 0,Y 47.1,Z 552.908,A -85,B 0,C 180,E1 -30113.354,E2 -30113.354} C_VEL
LIN {X 0,Y 43.509,Z 554.272,A -85,B 0,C 180,E1 -30121.013,E2 -30121.013} C_VEL
LIN {X 0,Y 39.35,Z 555.786,A -85,B 0,C 180,E1 -30139.711,E2 -30139.711} C_VEL
LIN {X 0,Y 38.798,Z 556.001,A -85,B 0,C 180,E1 -30149.999,E2 -30149.999} C_VEL
LIN {X 0,Y 39.348,Z 555.81,A -85,B 0,C 180,E1 -30160.288,E2 -30160.288} C_VEL
LIN {X 0,Y 43.496,Z 554.327,A -85,B 0,C 180,E1 -30178.994,E2 -30178.994} C_VEL
LIN {X 0,Y 47.081,Z 552.989,A -85,B 0,C 180,E1 -30186.661,E2 -30186.661} C_VEL
LIN {X 0,Y 53.695,Z 550.157,A -85,B 0,C 180,E1 -30196.044,E2 -30196.044} C_VEL
LIN {X 0,Y 61.275,Z 546.329,A -85,B 0,C 180,E1 -30203.405,E2 -30203.405} C_VEL
LIN {X 0,Y 70.956,Z 540.383,A -85,B 0,C 180,E1 -30210.314,E2 -30210.314} C_VEL
LIN {X 0,Y 75.211,Z 537.407,A -85,B 0,C 180,E1 -30212.587,E2 -30212.587} C_VEL
LIN {X 0,Y 76.676,Z 535.708,A -85,B 0,C 180,E1 -30216.431,E2 -30216.431} C_VEL
LIN {X 0,Y 78.516,Z 533.239,A -85,B 0,C 180,E1 -30224.423,E2 -30224.423} C_VEL
LIN {X 0,Y 79.66,Z 532.102,A -85,B 0,C 180,E1 -30229.837,E2 -30229.837} C_VEL
LIN {X 0,Y 80.669,Z 531.491,A -85,B 0,C 180,E1 -30235.002,E2 -30235.002} C_VEL
LIN {X 0,Y 81.51,Z 531.524,A -85,B 0,C 180,E1 -30240,E2 -30240} C_VEL
LIN {X 0,Y 80.726,Z 533.52,A -85,B 0,C 180,E1 -30245.228,E2 -30245.228} C_VEL
LIN {X 0,Y 79.681,Z 534.996,A -85,B 0,C 180,E1 -30247.12,E2 -30247.12} C_VEL
LIN {X 0,Y 77.906,Z 536.846,A -85,B 0,C 180,E1 -30248.589,E2 -30248.589} C_VEL
LIN {X 0,Y 75.231,Z 539.251,A -85,B 0,C 180,E1 -30249.917,E2 -30249.917} C_VEL
LIN {X 0,Y 66.721,Z 545.703,A -85,B 0,C 180,E1 -30253.39,E2 -30253.39} C_VEL
LIN {X 0,Y 59.221,Z 550.942,A -85,B 0,C 180,E1 -30258.308,E2 -30258.308} C_VEL
LIN {X 0,Y 51.916,Z 555.27,A -85,B 0,C 180,E1 -30263.961,E2 -30263.961} C_VEL
LIN {X 0,Y 42.134,Z 559.869,A -85,B 0,C 180,E1 -30273.488,E2 -30273.488} C_VEL
LIN {X 0,Y 37.246,Z 561.88,A -85,B 0,C 180,E1 -30280.997,E2 -30280.997} C_VEL
LIN {X 0,Y 30.545,Z 564.626,A -85,B 0,C 180,E1 -30302.603,E2 -30302.603} C_VEL
LIN {X 0,Y 29.318,Z 565.416,A -85,B 0,C 180,E1 -30316.132,E2 -30316.132} C_VEL
LIN {X 0,Y 29.745,Z 565.805,A -85,B 0,C 180,E1 -30330.001,E2 -30330.001} C_VEL
LIN {X 0,Y 30.534,Z 564.592,A -85,B 0,C 180,E1 -30357.41,E2 -30357.41} C_VEL
LIN {X 0,Y 37.237,Z 561.811,A -85,B 0,C 180,E1 -30379.022,E2 -30379.022} C_VEL
LIN {X 0,Y 44.804,Z 558.627,A -85,B 0,C 180,E1 -30389.626,E2 -30389.626} C_VEL
